(* POU Functions/F_GetVersionDehoff, ST *)
FUNCTION F_GetVersionDehoff : UINT
VAR_INPUT
	nVersionElement: INT := 0;
END_VAR
(*	Version history: This is for the program in the CX2020.  The HMI program version resisdes in the CP2612
Date	|	Rev	|	created under	|	Author				|	Remark		
---------------------------------------------------------------------------------------------------------------------------------------------------------------------
09/27/14	|	1.0	|	Build 2241	|	Ron Poehlmann		|	(Shipped on Machine #1 & 2)
12/04/14	|	1.1	|	Build 2241	|	Ron Poehlmann		|	Fixed problem caused by Fault History not being completed
															Added Fault Screen with Servo Axis Diagnostics #'s
															Moved into Persistent Data: U/X Axis Position and Speed variables & Tailstock Max Thrust
															Fixed Rung 117 to say 3B instead of 3A
															(* Remotely Installed on Machine #1 & #2*)
2/09/15	|	1.2	|	Build 2241	|	Ron Poehlmann		|	Changed Drill Cycle so that the Filter Fault does not stop the cycle.
															Worked on other Problems.
															(* Remotely Installed on Machine #2 & #1 *)
2/16/15	|	1.3	|	Build 2241	|	Ron Poehlmann		|	Rewrote Transfer Cycle.
															(* Remotely Installed on Machine #1 & #2 *)
2/18/15	|	1.3b	|											Fixed Reset of Servo Drives.
															(* Remotely Installed on Machine #1 & 2 *)
3/3/15	|	1.4	|	Build 2241	|	Ron Poehlmann		|	Added Recovery of Overtravel.
															Added checks and warnings before entering Auto.
															Added Single Homeing Button for WA, WB, and X Axis
															Modified Network Variables to assure alignment.
															Added Faults to Tailstock and Transfer.
															Shortened User name Passwords and added handshake bit.
															Added Recording of the W Axis Max Thrust Values.
															Added VFD Data Valid bit and Revised FB_EtherCAT_Emerson. 
7/8/15		Field mods										Added monitoring screen to CX to be able to view machie status.
															( Remotely Installed on Machine #1 - 4 )
11/05/15	|	1.5	|	Build 2241	|	Ron Poehlmann		|	Fixed typo that caused the X Axis Velocity not to be received from Panel B
															Added Fault condition to AC_CellRunoutFinish so it would Exit Auto on a Fault condition.
															Added Fault condition to AC_Init so it would Exit Auto on a Fault condition.
															Added Feed Over-ride as a setup feature.
															Fault at end of cycle if Lube Level Low Warning on for more than 2 cycles.
															Disable MPG if clamped.
															Fixed typo in FB_FixtureControl line 444 from nClampState to nUnclampState
															Changed Max Thrust Inputs for FB_Fixture Control
1/14/16	|	1.6	|	Build 2254	|	Ron Poehlmann		|	System Manager was Changed from V1 to V1.1 because of newer Card definitions.
															When Load Side switched - Swapp Load and unload Positions.
															Fixed a problem with the Waring 110 on Transfer_Cycle so that it will retriger in Cell Runout
																made step 10 check for bCellRunoutRequest.
*)
CASE nVersionElement OF
	1: F_GetVersionDehoff:=1;		(* Major Number *)
	2: F_GetVersionDehoff:=6;		(* ArboMex Program Revision Number *)
ELSE
	F_GetVersionDehoff:=16#FFFF;
END_CASE
END_FUNCTION

(* POU Programs/Build_Receive_Network_Data, ST *)
PROGRAM Build_Receive_Network_Data
VAR
	fbSideAUserNameInput: R_TRIG;			(* An User Name Input has just been received from Panel A *)
	fbSideBUserNameInput: R_TRIG;			(* An User Name Input has just been received from Panel B *)
	fbSideAPasswordInput: R_TRIG;				(* A Password Input has just been received from Panel A *)
	fbSideBPasswordInput: R_TRIG;				(* A Password Input has just been received from Panel B *)
	fbSideASavePasswordInputTrig: R_TRIG;		(* A Save Password Input has just been received from Panel A *)
	fbSideBSavePasswordInput: R_TRIG;		(* A Save Password Input has just been received from Panel B *)
	fbSideAEnableRTrig: R_TRIG;
	fbSideBEnableRTrig: R_TRIG;
	fbTestSpeedActiveRTrig: R_TRIG;			(* Push Button pressed to Activate/Deactivate the Test Speed *)
	nTest: INT := 0;		(* Test Counter*)
	fUAxisLoadPositionTempVariable: LREAL := 0.0;		(*A Temp variable used to swap the Load and unload position*)
END_VAR
(* Login Varialbes *)
(* If the Login PB or Logout PB is pressed on either screen, then turn on the bit*)
bLoginPB := stReceivePanelA.arrBOOL[8] OR stReceivePanelB.arrBOOL[8];
bLogoutPB := stReceivePanelA.arrBOOL[9] OR stReceivePanelB.arrBOOL[9];

(* Receive the User ID Input *)
(* Only place what is received into the Username when the received value first changes
	Also if they enter a wrong value, then we want to trigger when it changes. 
	When we see a change from '' set the handshake bit.  
		The Panel will then set the variable to '' again, so turn off the handshake bit.*)
fbSideAUserNameInput(CLK:=stReceivePanelA.arrTEXTSTRING[2] <> '');
fbSideBUserNameInput(CLK:=stReceivePanelB.arrTEXTSTRING[2] <> '');
IF fbSideAUserNameInput.Q THEN
	bUserNameHandshake:=TRUE;
	sUsername := stReceivePanelA.arrTEXTSTRING[2];
ELSIF fbSideBUserNameInput.Q THEN
	bUserNameHandshake:=TRUE;
	sUsername := stReceivePanelB.arrTEXTSTRING[2];
ELSIF (stReceivePanelA.arrTEXTSTRING[2] = '') AND (stReceivePanelB.arrTEXTSTRING[2] = '') THEN
	bUserNameHandshake:=FALSE;
END_IF

(* Receive the Password Input *)
fbSideAPasswordInput(CLK:=stReceivePanelA.arrTEXTSTRING[3] <> '');
fbSideBPasswordInput(CLK:=stReceivePanelB.arrTEXTSTRING[3] <> '');
IF fbSideAPasswordInput.Q THEN
	bPasswordHandshake:=TRUE;
	sPassword := stReceivePanelA.arrTEXTSTRING[3];
ELSIF fbSideBPasswordInput.Q THEN
	bPasswordHandshake:=TRUE;
	sPassword := stReceivePanelB.arrTEXTSTRING[3];
ELSIF (stReceivePanelA.arrTEXTSTRING[3] = '') AND (stReceivePanelB.arrTEXTSTRING[3] = '') THEN
	bPasswordHandshake:=FALSE;
END_IF

(* Receive the Save Password Input *)
fbSideASavePasswordInputTrig(CLK:=stReceivePanelA.arrTEXTSTRING[4] <> '');
fbSideBSavePasswordInput(CLK:=stReceivePanelB.arrTEXTSTRING[4] <> '');
IF (stReceivePanelA.arrTEXTSTRING[4] <> '') THEN
	IF stReceivePanelA.arrTEXTSTRING[4]=sPasswordSupervisorUC OR
		stReceivePanelA.arrTEXTSTRING[4]=sPasswordSupervisor OR
		stReceivePanelA.arrTEXTSTRING[4]=sPasswordSuperUC OR
		stReceivePanelA.arrTEXTSTRING[4]=sPasswordSuper
	THEN
		bWrongSavePassword:=FALSE;
		bSavePasswordHandshake:=TRUE;
		sSavePassword := stReceivePanelA.arrTEXTSTRING[4];
	(* Password is not correct *)
	ELSE
		bWrongSavePassword:=TRUE;
	END_IF
END_IF
IF (stReceivePanelB.arrTEXTSTRING[4] <> '') THEN
	IF stReceivePanelB.arrTEXTSTRING[4]=sPasswordSupervisorUC OR
		stReceivePanelB.arrTEXTSTRING[4]=sPasswordSupervisor OR
		stReceivePanelA.arrTEXTSTRING[4]=sPasswordSuperUC OR
		stReceivePanelA.arrTEXTSTRING[4]=sPasswordSuper
	THEN
		bWrongSavePassword:=FALSE;
		bSavePasswordHandshake:=TRUE;
		sSavePassword := stReceivePanelB.arrTEXTSTRING[4];
		(* Password is not correct *)
	ELSE
		bWrongSavePassword:=TRUE;
	END_IF
END_IF
IF (stReceivePanelA.arrTEXTSTRING[4] = '') AND (stReceivePanelB.arrTEXTSTRING[4] = '') THEN
	bSavePasswordHandshake:=FALSE;
	bWrongSavePassword:=FALSE;
END_IF


(* Call Actions *)
Auto_Screen_Receive;
Part_Program_Screen;
Transfer_Screen;
Fixture_Screen;
Secret_Screen;
Test_Speed_Screen;
Manual_Screen_Receive;
END_PROGRAM
ACTION Auto_Screen_Receive:
(* Push Buttons *)
bEnterManualModePB := 	stReceivePanelA.arrBOOL[1] OR stReceivePanelB.arrBOOL[1];
bEnterAutoModePB := 		stReceivePanelA.arrBOOL[2] OR stReceivePanelB.arrBOOL[2];
bResetCycleCounterPB := 	stReceivePanelA.arrBOOL[3] OR stReceivePanelB.arrBOOL[3];;
bFaultResetPB := 			stReceivePanelA.arrBOOL[4] OR stReceivePanelB.arrBOOL[4];
bResetTotalCountPB := 	stReceivePanelA.arrBOOL[5] OR stReceivePanelB.arrBOOL[5];
bCellRunOutPB := 			stReceivePanelA.arrBOOL[67] OR stReceivePanelB.arrBOOL[67];
bResetA1CountPB:= 		stReceivePanelA.arrBOOL[42] OR stReceivePanelB.arrBOOL[42];
bResetA2CountPB:= 		stReceivePanelA.arrBOOL[43] OR stReceivePanelB.arrBOOL[43];
bResetA3CountPB:= 		stReceivePanelA.arrBOOL[44] OR stReceivePanelB.arrBOOL[44];
bResetB1CountPB:= 		stReceivePanelA.arrBOOL[45] OR stReceivePanelB.arrBOOL[45];
bResetB2CountPB:= 		stReceivePanelA.arrBOOL[46] OR stReceivePanelB.arrBOOL[46];
bResetB3CountPB:= 		stReceivePanelA.arrBOOL[47] OR stReceivePanelB.arrBOOL[47];
END_ACTION
ACTION Fixture_Screen:
(* Fixture common Inputs *)
(* When a Transfer position Input is received from Panel A or B then modify *)
IF stReceivePanelA.arrLREAL[20] <> 0.0 THEN
	fWAxisTransferPosition :=stReceivePanelA.arrLREAL[20];
ELSIF stReceivePanelB.arrLREAL[20] <> 0.0 THEN
	fWAxisTransferPosition :=stReceivePanelB.arrLREAL[20];
END_IF

(* When a Drill Position Input is received from Panel A or B then modify *)
IF stReceivePanelA.arrLREAL[21] <> 0.0 THEN
	fWAxisDrillPosition :=stReceivePanelA.arrLREAL[21];
ELSIF stReceivePanelB.arrLREAL[21] <> 0.0 THEN
	fWAxisDrillPosition :=stReceivePanelB.arrLREAL[21];
END_IF

(* A Side *)
(*Push Buttons Side A *)
bWAAxisHomePB := stReceivePanelA.arrBOOL[30];
bWAAxisAdvancePB := stReceivePanelA.arrBOOL[31];
bWAAxisRetractPB := stReceivePanelA.arrBOOL[32];
bAColletClosePB := stReceivePanelA.arrBOOL[33];
bAColletOpenPB := stReceivePanelA.arrBOOL[34];
bAEjectorsAdvancePB := stReceivePanelA.arrBOOL[35];
bAEjectorsRetractPB := stReceivePanelA.arrBOOL[36];

	(* B Side *)
(*Push Buttons Side B *)
bWBAxisHomePB := stReceivePanelB.arrBOOL[30];
bWBAxisAdvancePB := stReceivePanelB.arrBOOL[31];
bWBAxisRetractPB := stReceivePanelB.arrBOOL[32];
bBColletClosePB := stReceivePanelB.arrBOOL[33];
bBColletOpenPB := stReceivePanelB.arrBOOL[34];
bBEjectorsAdvancePB := stReceivePanelB.arrBOOL[35];
bBEjectorsRetractPB := stReceivePanelB.arrBOOL[36];

(* If We have a FAULT we do not want to permit manual operations.
	So turn off any PB bits that may have been pushed. *)
IF bMachineFault
	OR nAutoCycleStep=AC_Drill
	OR nAutoCycleStep=AC_DrillReturn
	OR nAutoCycleStep=AC_Retract
THEN
	bWAAxisHomePB := FALSE;
	bWAAxisAdvancePB := FALSE;
	bWAAxisRetractPB := FALSE;
	bAColletClosePB := FALSE;
	bAColletOpenPB := FALSE;
	bAEjectorsAdvancePB := FALSE;
	bAEjectorsRetractPB := FALSE;
	bWBAxisHomePB := FALSE;
	bWBAxisAdvancePB := FALSE;
	bWBAxisRetractPB := FALSE;
	bBColletClosePB := FALSE;
	bBColletOpenPB := FALSE;
	bBEjectorsAdvancePB := FALSE;
	bBEjectorsRetractPB := FALSE;
END_IF
END_ACTION
ACTION Manual_Screen_Receive:
(* MANUAL SCREEN *)

(* Push Buttons *)
(* When the Start Hydraulic PB is pressed on either panel *)
bStartHydraulicPB := stReceivePanelA.arrBOOL[60] OR stReceivePanelB.arrBOOL[60];
(* When the Stop Hydraulic PB is pressed on either panel *)
bStopHydraulicPB := stReceivePanelA.arrBOOL[61] OR stReceivePanelB.arrBOOL[61];
(* When the Start Coolant PB is pressed on either panel *)
bCoolantStartPB := stReceivePanelA.arrBOOL[62] OR stReceivePanelB.arrBOOL[62];
(* When the Stop Coolant PB is pressed on either panel *)
bCoolantStopPB := stReceivePanelA.arrBOOL[63] OR stReceivePanelB.arrBOOL[63];
(* Setup is dependant on the side it is Pressed *)
bEnterSetupPB_A := stReceivePanelA.arrBOOL[64];
bEnterSetupPB_B := stReceivePanelB.arrBOOL[64];
(* Set Zero is dependant on the side it is Pressed *)
bSetZeroPositionPB_A := stReceivePanelA.arrBOOL[65];
bSetZeroPositionPB_B := stReceivePanelB.arrBOOL[65];
(* Move To Zero is dependant on the side it is Pressed *)
bMoveToZeroPositionPB_A := stReceivePanelA.arrBOOL[66];
bMoveToZeroPositionPB_B := stReceivePanelB.arrBOOL[66];

(* When the Home All Automation PB is pressed on either panel *)
bHomeAutomationPB := stReceivePanelA.arrBOOL[68] OR stReceivePanelB.arrBOOL[68];
END_ACTION
ACTION Part_Program_Screen:
(* PART PROGRAM Inputs *)

(*  Change the Part Program Name when Inserted by operator *)
IF stReceivePanelA.arrTEXTSTRING[1] <> ''  THEN
	sPartProgramName := stReceivePanelA.arrTEXTSTRING[1];
ELSIF stReceivePanelB.arrTEXTSTRING[1] <> '' THEN
	sPartProgramName := stReceivePanelB.arrTEXTSTRING[1];
END_IF

(* Save Part Progarm Push Button *)
bPartProgramSavePB:= stReceivePanelA.arrBOOL[11] OR stReceivePanelB.arrBOOL[11];

(* Leave the PP_SAVE screen *)
IF stReceivePanelA.arrBOOL[69] OR stReceivePanelB.arrBOOL[69] THEN
	sSavePassword:='';
END_IF


(* Load Part Program Push Button - Not available in Auto  *)
bPartProgramLoadPB := stReceivePanelA.arrBOOL[12] OR stReceivePanelB.arrBOOL[12];

(**** IMPORTANT! ***  If the system is in AUTO or In Cycle we need to send a Warning  *)

(* Toggle the state of Spindle Retract mode when PB received from panels *)
IF stReceivePanelA.arrBOOL[10] OR stReceivePanelB.arrBOOL[10] THEN
	IF bSpindleRetractMode THEN
		bSpindleRetractMode:=FALSE;
	ELSE bSpindleRetractMode:=TRUE;
	END_IF
END_IF

(* When a Start Feed Input is received from either panel then modify *)
IF stReceivePanelA.arrLREAL[1] > 0.0 THEN
	fStartFeed:=stReceivePanelA.arrLREAL[1];
ELSIF stReceivePanelB.arrLREAL[1] > 0.0 THEN
	fStartFeed:=stReceivePanelB.arrLREAL[1];
END_IF

(* When a Start Feed Input is received from either panel then modify *)
IF stReceivePanelA.arrLREAL[2] > 0.0 THEN
	fFinishFeed:=stReceivePanelA.arrLREAL[2];
ELSIF stReceivePanelB.arrLREAL[2] > 0.0 THEN
	fFinishFeed:=stReceivePanelB.arrLREAL[2];
END_IF

(* When a Start Depth Input is received from either panel then modify *)
IF stReceivePanelA.arrLREAL[3] < 0.0 THEN
	fStartDepth:=stReceivePanelA.arrLREAL[3];
ELSIF stReceivePanelB.arrLREAL[3] < 0.0 THEN
	fStartDepth:=stReceivePanelB.arrLREAL[3];
END_IF

(* When a Finish Depth Input is received from either panel then modify *)
IF stReceivePanelA.arrLREAL[4] < 0.0 THEN
	fFinishDepth:=stReceivePanelA.arrLREAL[4];
ELSIF stReceivePanelB.arrLREAL[4] < 0.0 THEN
	fFinishDepth:=stReceivePanelB.arrLREAL[4];
END_IF

(* When a Dwell Time Input is received from either panel then modify *)
IF stReceivePanelA.arrLREAL[5] > 0.0 THEN
	fDwellTime:=stReceivePanelA.arrLREAL[5];
ELSIF stReceivePanelB.arrLREAL[5] > 0.0 THEN
	fDwellTime:=stReceivePanelB.arrLREAL[5];
END_IF

(* When a Retract Rate Input is received from either panel then modify *)
IF stReceivePanelA.arrLREAL[6] > 0.0 THEN
	fRetractRate:=stReceivePanelA.arrLREAL[6];
ELSIF stReceivePanelB.arrLREAL[6] > 0.0 THEN
	fRetractRate:=stReceivePanelB.arrLREAL[6];
END_IF

(* When a fDrill Tip Offset Input is received from either panel then modify *)
IF stReceivePanelA.arrLREAL[7] > 0.0 THEN
	fDrillTipOffset:=stReceivePanelA.arrLREAL[7];
ELSIF stReceivePanelB.arrLREAL[7] > 0.0 THEN
	fDrillTipOffset:=stReceivePanelB.arrLREAL[7];
END_IF

(* When a RPM Request Input is received from either panel then modify *)
IF stReceivePanelA.arrLREAL[8] > 0.0 THEN
	fRPMRequest:=stReceivePanelA.arrLREAL[8];
ELSIF stReceivePanelB.arrLREAL[8] > 0.0 THEN
	fRPMRequest:=stReceivePanelB.arrLREAL[8];
END_IF

(* When a Tool Diameter Input is received from either panel then modify *)
IF stReceivePanelA.arrLREAL[9] > 0.0 THEN
	fToolDiameter:=stReceivePanelA.arrLREAL[9];
ELSIF stReceivePanelB.arrLREAL[9] > 0.0 THEN
	fToolDiameter:=stReceivePanelB.arrLREAL[9];
END_IF

(* When a Coolant Pressure Input is received from either panel then modify *)
IF stReceivePanelA.arrLREAL[10] > 0.0 THEN
	fCoolantPressure:=stReceivePanelA.arrLREAL[10];
ELSIF stReceivePanelB.arrLREAL[10] > 0.0 THEN
	fCoolantPressure:=stReceivePanelB.arrLREAL[10];
END_IF

(* When a Coolant Flow Max Input is received from either panel then modify *)
IF stReceivePanelA.arrLREAL[11] > 0.0 THEN
	fCoolantFlowMax:=stReceivePanelA.arrLREAL[11];
ELSIF stReceivePanelB.arrLREAL[11] > 0.0 THEN
	fCoolantFlowMax:=stReceivePanelB.arrLREAL[11];
END_IF

(* When a Coolant Flow Min Input is received from either panel then modify *)
IF stReceivePanelA.arrLREAL[12] > 0.0 THEN
	fCoolantFlowMin:=stReceivePanelA.arrLREAL[12];
ELSIF stReceivePanelB.arrLREAL[12] > 0.0 THEN
	fCoolantFlowMin:=stReceivePanelB.arrLREAL[12];
END_IF

(* When Max cycles Set is received from either panel then modify *)
IF stReceivePanelA.arrUDINTIGER[1] > 0 THEN
	nMaxCycles := stReceivePanelA.arrUDINTIGER[1];
ELSIF  stReceivePanelB.arrUDINTIGER[1] > 0 THEN
	nMaxCycles := stReceivePanelB.arrUDINTIGER[1];
END_IF

(* When Spindle Load Max Set is received from either panel then modify *)
IF stReceivePanelA.arrUDINTIGER[2] > 0 THEN
	nSpindleLoadMax := stReceivePanelA.arrUDINTIGER[2];
ELSIF  stReceivePanelB.arrUDINTIGER[2] > 0 THEN
	nSpindleLoadMax := stReceivePanelB.arrUDINTIGER[2];
END_IF

(* When Servo Thrust Max Set is received from either panel then modify *)
IF stReceivePanelA.arrUDINTIGER[3] > 0 THEN
	nServoThrustMax := stReceivePanelA.arrUDINTIGER[3];
ELSIF  stReceivePanelB.arrUDINTIGER[3] > 0 THEN
	nServoThrustMax := stReceivePanelB.arrUDINTIGER[3];
END_IF
END_ACTION
ACTION Secret_Screen:
(* Receive the PB's from the Panels *)
(* The Panels Make sure you must not be in Auto Mode *)
IF stReceivePanelA.arrBOOL[6] OR stReceivePanelB.arrBOOL[6] THEN
	bASideIsLoadPB := TRUE;
ELSIF  stReceivePanelA.arrBOOL[7] OR stReceivePanelB.arrBOOL[7] THEN
	bBSideIsLoadPB := TRUE;
END_IF

fbSideAEnableRTrig(CLK:=stReceivePanelA.arrBOOL[40] OR stReceivePanelB.arrBOOL[40]);
IF fbSideAEnableRTrig.Q THEN
	IF bSideAEnabled THEN
		bSideAEnabled := FALSE;
	ELSE
		bSideAEnabled :=TRUE;
	END_IF
END_IF

fbSideBEnableRTrig(CLK:=stReceivePanelA.arrBOOL[41] OR stReceivePanelB.arrBOOL[41]);
IF fbSideBEnableRTrig.Q THEN
	IF bSideBEnabled THEN
		bSideBEnabled := FALSE;
	ELSE
		bSideBEnabled :=TRUE;
	END_IF
END_IF

IF bASideIsLoadPB THEN
	sLoadSideSet := 'A';
	(* Swap the Load and Unload Positions *)
	fUAxisLoadPositionTempVariable:=fUAxisLoadSidePosition;
	fUAxisLoadSidePosition:= fUAxisUnloadSidePosition;
	fUAxisUnloadSidePosition:=fUAxisLoadPositionTempVariable;
	bASideIsLoadPB := FALSE;
ELSIF bBSideIsLoadPB THEN
	sLoadSideSet :='B';
	(* Swap the Load and Unload Positions *)
	fUAxisLoadPositionTempVariable:=fUAxisLoadSidePosition;
	fUAxisLoadSidePosition:= fUAxisUnloadSidePosition;
	fUAxisUnloadSidePosition:=fUAxisLoadPositionTempVariable;
	bBSideIsLoadPB := FALSE;
END_IF

IF (stReceivePanelA.arrUDINTIGER[10] >0) THEN
	nUAxisThrustMax := stReceivePanelA.arrUDINTIGER[10];
ELSIF (stReceivePanelB.arrUDINTIGER[10] >0) THEN
	nUAxisThrustMax := stReceivePanelB.arrUDINTIGER[10];
END_IF

(* Tailstock Torque Limit During Clamping *)
IF (stReceivePanelA.arrUDINTIGER[11] >0) THEN
	nTailstockClampingTorqueLimit := UDINT_TO_INT(stReceivePanelA.arrUDINTIGER[11]);
ELSIF (stReceivePanelB.arrUDINTIGER[11] >0) THEN
	nTailstockClampingTorqueLimit := UDINT_TO_INT(stReceivePanelB.arrUDINTIGER[11]);
END_IF

(* Receive the WA Axis Home Offset *)
(* Must compare with current value because 0.0 is an option *)
IF stReceivePanelA.arrLREAL[17] <> 0.0  THEN
	fWAAxisHomeOffset := stReceivePanelA.arrLREAL[17];
ELSIF stReceivePanelB.arrLREAL[17] <> 0.0 THEN
	fWAAxisHomeOffset := stReceivePanelB.arrLREAL[17];
END_IF

(* Receive the WB Axis Home Offset *)
IF stReceivePanelA.arrLREAL[18] <> 0.0  THEN
	fWBAxisHomeOffset := stReceivePanelA.arrLREAL[18];
ELSIF stReceivePanelB.arrLREAL[18] <> 0.0 THEN
	fWBAxisHomeOffset := stReceivePanelB.arrLREAL[18];
END_IF

(* Receive the W Axis Amount to Move Off of Bushing *)
IF stReceivePanelA.arrLREAL[19] <> 0.0 THEN
	fWAxisMoveOffBushing :=stReceivePanelA.arrLREAL[19];
ELSIF stReceivePanelB.arrLREAL[19] <> 0.0 THEN
	fWAxisMoveOffBushing :=stReceivePanelB.arrLREAL[19];
END_IF

(* Receive the W Axis Move Velocity *)
IF stReceivePanelA.arrLREAL[24] > 0.0 THEN
	fTailstockVelocity :=stReceivePanelA.arrLREAL[24];
ELSIF stReceivePanelB.arrLREAL[24] > 0.0 THEN
	fTailstockVelocity :=stReceivePanelB.arrLREAL[24];
END_IF

(* When a WA Axis Max Thrust Input is received from Panel A then modify *)
IF stReceivePanelA.arrUDINTIGER[5] > 0.0 THEN
	nWAAxisThrustMax :=stReceivePanelA.arrUDINTIGER[5];
ELSIF stReceivePanelB.arrUDINTIGER[5] > 0.0 THEN
	nWAAxisThrustMax :=stReceivePanelB.arrUDINTIGER[5];
END_IF

(* When a WB Axis Max Thrust Input is received from Panel B then modify *)
IF stReceivePanelA.arrUDINTIGER[6] > 0.0 THEN
	nWBAxisThrustMax :=stReceivePanelA.arrUDINTIGER[6];
ELSIF stReceivePanelB.arrUDINTIGER[6] > 0.0 THEN
	nWBAxisThrustMax :=stReceivePanelB.arrUDINTIGER[6];
END_IF
END_ACTION
ACTION Test_Speed_Screen:
(* Test Speed  Screen *)
(* The Test Speed would be like a feed over-ride and changes the speeds of the WA, WB and X Axis movements *)

(* When either panel sets the  "Test Speed Input" then make it Current Test Speed *)
IF (stReceivePanelA.arrUDINTIGER[15] <> 0.0) THEN
	nTestSpeedOverRide := stReceivePanelA.arrUDINTIGER[15];
ELSIF (stReceivePanelB.arrUDINTIGER[15] <> 0.0) THEN
	nTestSpeedOverRide := stReceivePanelB.arrUDINTIGER[15];
END_IF

(* When the Test Speed Overide PB is pressed on either screen, we toggle the state On/Off *)
fbTestSpeedActiveRTrig(CLK:=stReceivePanelA.arrBOOL[15] OR stReceivePanelB.arrBOOL[15]);
IF fbTestSpeedActiveRTrig.Q THEN
	IF bTestSpeedOn THEN
		bTestSpeedOn := FALSE;
	ELSE
		bTestSpeedOn := TRUE;
	END_IF
END_IF

(* When the Test Speed is Activated we want to Change the velocities that we feed to the Axis Move FB's *)
IF bTestSpeedOn THEN
	fWAxisFastVelocity := fTailstockVelocity * (nTestSpeedOverRide/100.0);
	fWAxisClampVelocity :=  fTailstockClampVelocity * (nTestSpeedOverRide/100.0);
	fTransferMoveVelo := fUAxisVelocity  * (nTestSpeedOverRide/100.0);
ELSE
	fWAxisFastVelocity := fTailstockVelocity;
	fWAxisClampVelocity :=  fTailstockClampVelocity;
	fTransferMoveVelo:=  fUAxisVelocity;
END_IF
END_ACTION
ACTION Transfer_Screen:
(* TRANSFER Screen Inputs *)

(* Raise and Lower Push Buttons *)
bTransferUpPB := (stReceivePanelA.arrBOOL[20] OR stReceivePanelB.arrBOOL[20]);
bTransferDownPB := (stReceivePanelA.arrBOOL[21] OR stReceivePanelB.arrBOOL[21]);

(* Home U Axis PB *)
bHomeUAxisPB := (stReceivePanelA.arrBOOL[22] OR stReceivePanelB.arrBOOL[22]);

(* Move U Axis PB's *)
bMoveUtoLoadPB := (stReceivePanelA.arrBOOL[23] OR stReceivePanelB.arrBOOL[23]);
bMoveUtoUnloadPB := (stReceivePanelA.arrBOOL[24] OR stReceivePanelB.arrBOOL[24]);

(* When we have a FAULT we want to disable manual functions.
	So turn off any PB's that could have been pushed *) 
IF bMachineFault
	OR nAutoCycleStep=AC_Drill
	OR nAutoCycleStep=AC_DrillReturn
	OR nAutoCycleStep=AC_Retract
THEN
	bTransferUpPB := FALSE;
	bTransferDownPB := FALSE;
	bHomeUAxisPB:= FALSE;
	bMoveUtoLoadPB:= FALSE;
	bMoveUtoUnloadPB:= FALSE;
END_IF

(* When either side sets the U Axis A Side position then put it in appropriate Load or Unload variable *)
IF (stReceivePanelA.arrLREAL[15] <>0) THEN	(* fUAxisASidePositionInput *)
	IF (sLoadSideSet = 'A') THEN
		fUAxisLoadSidePosition := stReceivePanelA.arrLREAL[15];
	ELSIF (sLoadSideSet = 'B') THEN
		fUAxisUnloadSidePosition := stReceivePanelA.arrLREAL[15];
	ELSE
		bLoadSideNotSelected := TRUE;
	END_IF
ELSIF (stReceivePanelB.arrLREAL[15] <>0) THEN	(* fUAxisASidePositionInput *)
	IF (sLoadSideSet = 'A') THEN
		fUAxisLoadSidePosition := stReceivePanelB.arrLREAL[15];
	ELSIF (sLoadSideSet = 'B') THEN
		fUAxisUnloadSidePosition := stReceivePanelB.arrLREAL[15];
	ELSE
		bLoadSideNotSelected := TRUE;
	END_IF
END_IF

(* When either side sets the U Axis B Side position then put it in appropriate Load or Unload variable *)
IF (stReceivePanelA.arrLREAL[16] <> 0.0) THEN	(* fUAxisBSidePositionInput *)
	IF (sLoadSideSet = 'A') THEN
		fUAxisUnloadSidePosition := stReceivePanelA.arrLREAL[16];
	ELSIF (sLoadSideSet = 'B') THEN
		fUAxisLoadSidePosition := stReceivePanelA.arrLREAL[16];
	ELSE
		bLoadSideNotSelected := TRUE;
	END_IF
ELSIF (stReceivePanelB.arrLREAL[16] <> 0.0) THEN	(* fUAxisBSidePositionInput *)
	IF (sLoadSideSet = 'A') THEN
		fUAxisUnloadSidePosition := stReceivePanelB.arrLREAL[16];
	ELSIF (sLoadSideSet = 'B') THEN
		fUAxisLoadSidePosition := stReceivePanelB.arrLREAL[16];
	ELSE
		bLoadSideNotSelected := TRUE;
	END_IF
END_IF

(* When either side sets the U Axis "Transfer Speed" then make it Current Speed *)
IF (stReceivePanelA.arrLREAL[25] <> 0.0) THEN
	fUAxisVelocity := stReceivePanelA.arrLREAL[25];
ELSIF (stReceivePanelB.arrLREAL[25] <> 0.0) THEN
	fUAxisVelocity := stReceivePanelB.arrLREAL[25];
END_IF
END_ACTION

(* POU Programs/P_PartProgramStorage, ST *)
PROGRAM P_PartProgramStorage
VAR
	fbPartProgramSaveRTRIG: R_TRIG;			(* Trigger for Part Program Save PB *)
	fbPartProgramLoadRTRIG: R_TRIG;			(* Trigger for Part Program Load PB *)
	bSave: BOOL := FALSE;
	bLoad: BOOL := FALSE;
	bFailed: BOOL := FALSE;
	bSuccess: BOOL := FALSE;

	(* Function Blocks w/ Helpers *)
	fbFileOpen: FB_FileOpen;
	bFileOpen: BOOL := FALSE;
	fbFileClose: FB_FileClose;
	nOpenType: DWORD;
	bFileClose: BOOL := FALSE;
	fbFilePuts: FB_FilePuts;
	bFilePuts: BOOL := FALSE;
	fbFileGets: FB_FileGets;
	bFileGets: BOOL := FALSE;
	hFileHandle: UINT := 0;
	sFileName: T_MaxString := '';

	(* State Variables *)
	nStep: USINT := 0;

	(* Read Variables  Note: if size changes it must be changed here and in the program below *)
	arrDataRead: ARRAY [1..25] OF T_MaxString;
	nReadCount: USINT := 0;

	(* Write Variables *)
	arrDataWrite: ARRAY [1..25] OF T_MaxString;
	nWriteCount: USINT := 0;

	nTestCount: INT := 0;		(* Test Counter *)
	bTestbit1: BOOL := FALSE;		(* Test Bit *)
END_VAR
fbPartProgramSaveRTRIG(CLK:= bPartProgramSavePB);
fbPartProgramLoadRTRIG(CLK:= bPartProgramLoadPB);

IF fbPartProgramSaveRTRIG.Q AND NOT(bSave OR bLoad) THEN
	(* When the Yes PB is pressed then check the password input *)
	IF sSavePassword=sPasswordSupervisorUC OR
		sSavePassword=sPasswordSupervisor OR
		sSavePassword=sPasswordSuperUC OR
		sSavePassword=sPasswordSuper
	THEN	(* Reset Values *)
		bFailed:=FALSE;
		bSuccess:=FALSE;
		sFileOpError:='';
		bSave:=TRUE;
		sSavePassword:='';
	END_IF
ELSIF fbPartProgramLoadRTRIG.Q AND NOT(bSave OR bLoad) THEN
	bFailed:=FALSE;
	sFileOpError:='';
	bSuccess:=FALSE;
	bLoad:=TRUE;
END_IF

sFileName:=CONCAT('\Hard Disk\ftp\',CONCAT(sPartProgramName, '.CSV'));


(* Load Part Program *)
IF bLoad AND NOT(bSave) THEN
	CASE nStep OF
	0:(* Open File *)
		nOpenType:=FOPEN_MODEREAD;
		(*ERROR*)
		IF bFileOpen AND fbFileOpen.bError THEN
			bFileOpen:=FALSE;
			bLoad:=FALSE;
			bFailed:=TRUE;
			sFileOpError:=CONCAT('Open Error:  ',UDINT_TO_STRING(fbFileOpen.nErrId));
		ELSIF bFileOpen AND NOT(fbFileOpen.bBusy) THEN
			bFileOpen:=FALSE;
			nReadCount:=1;
			nStep:=nStep+1;
		END_IF
		bFileOpen:=TRUE;

	1:(* Read File *)
		IF (nReadCount<=25) OR NOT(fbFileGets.bEOF) THEN
			(*ERROR*)
			IF bFileGets AND fbFileGets.bError THEN
				nStep:=nStep+1;
				bFailed:=TRUE;
				sFileOpError:=CONCAT('Read Error:  ',UDINT_TO_STRING(fbFileGets.nErrId));
			ELSIF bFileGets AND NOT(fbFileGets.bBusy) THEN
				arrDataRead[nReadCount]:=fbFileGets.sLine;
				bFileGets:=FALSE;
				nReadCount:=nReadCount+1;
			ELSIF NOT(bFileGets) THEN
				bFileGets:=TRUE;
			END_IF
		END_IF
		IF nReadCount>25 THEN
			nStep:=nStep+1;
		END_IF

	2:(* Close File *)
		(*ERROR*)
		IF bFileClose AND fbFileClose.bError THEN
			sFileOpError:=CONCAT('Close Error:  ',UDINT_TO_STRING(fbFileClose.nErrId));
			bFileClose:=FALSE;
			bLoad:=FALSE;
			bFailed:=TRUE;
		ELSIF bFileClose AND NOT(fbFileClose.bBusy) THEN
			bFileClose:=FALSE;
			IF bFailed THEN
				bLoad:=FALSE;
			ELSE
				nStep:=nStep+1;
			END_IF
		END_IF
		bFileClose:=TRUE;

	3:(* Convert Data / Done *)
		fStartFeed				:= STRING_TO_LREAL(arrDataRead[2]);
		fFinishFeed 				:= STRING_TO_LREAL(arrDataRead[3]);
		fStartDepth 				:= STRING_TO_LREAL(arrDataRead[4]);
		fFinishDepth 				:= STRING_TO_LREAL(arrDataRead[5]);
		fDwellTime 				:= STRING_TO_LREAL(arrDataRead[6]);
		fRetractRate 				:= STRING_TO_LREAL(arrDataRead[7]);
		fDrillTipOffset				:= STRING_TO_LREAL(arrDataRead[8]);
		fRPMRequest			:= STRING_TO_LREAL(arrDataRead[9]);
		fToolDiameter			:= STRING_TO_LREAL(arrDataRead[10]);
		fCoolantPressure			:= STRING_TO_LREAL(arrDataRead[11]);
		fCoolantFlowMax			:= STRING_TO_LREAL(arrDataRead[12]);
		fCoolantFlowMin			:= STRING_TO_LREAL(arrDataRead[13]);
		nMaxCycles				:= LREAL_TO_UDINT(STRING_TO_LREAL(arrDataRead[14]));
		fWAxisTransferPosition		:= STRING_TO_LREAL(arrDataRead[15]);
		fWAxisDrillPosition		:= STRING_TO_LREAL(arrDataRead[16]);
		fWAxisMoveOffBushing		:= STRING_TO_LREAL(arrDataRead[17]);
		(*	:= STRING_TO_LREAL(arrDataRead[18]);		*)
		bSpindleRetractMode		:= STRING_TO_BOOL(arrDataRead[19]);
		nSpindleLoadMax			:= LREAL_TO_UDINT(STRING_TO_LREAL(arrDataRead[20]));
		nServoThrustMax			:= LREAL_TO_UDINT(STRING_TO_LREAL(arrDataRead[21]));
		(*	:=STRING_TO_LREAL(arrDataRead[22]);		*)
		(*	:=STRING_TO_LREAL(arrDataRead[23]);		*)
		(*	:=STRING_TO_LREAL(arrDataRead[24]);		*)
		(*	:=STRING_TO_LREAL(arrDataRead[25]);		*)
		(* IF MORE THAN 25 VARIABLES
			THEN MUST CHANGE nReadCount COMPARASONS IN nStep 1 *)
		nStep:=nStep+1;

	4:(* Done *)
		nStep:=0;
		bLoad:=FALSE;
		bSuccess:=TRUE;
		sLastLoadedPartProgramName := sPartProgramName;
		sCurrentPartProgram := sPartProgramName;

	END_CASE


ELSIF bSave AND NOT(bLoad) THEN
	CASE nStep OF
	0:(* Prepare Data *)
		arrDataWrite[1]	:= CONCAT(sPartProgramName,'$L');
		arrDataWrite[2]	:= CONCAT(LREAL_TO_STRING(fStartFeed),'$L');
		arrDataWrite[3]	:= CONCAT(LREAL_TO_STRING(fFinishFeed),'$L');
		arrDataWrite[4]	:= CONCAT(LREAL_TO_STRING(fStartDepth),'$L');
		arrDataWrite[5]	:= CONCAT(LREAL_TO_STRING(fFinishDepth),'$L');
		arrDataWrite[6]	:= CONCAT(LREAL_TO_STRING(fDwellTime),'$L');
		arrDataWrite[7]	:= CONCAT(LREAL_TO_STRING(fRetractRate),'$L');
		arrDataWrite[8]	:= CONCAT(LREAL_TO_STRING(fDrillTipOffset),'$L');
		arrDataWrite[9]	:= CONCAT(LREAL_TO_STRING(fRPMRequest),'$L');
		arrDataWrite[10]	:= CONCAT(LREAL_TO_STRING(fToolDiameter),'$L');
		arrDataWrite[11]	:= CONCAT(LREAL_TO_STRING(fCoolantPressure),'$L');
		arrDataWrite[12]	:= CONCAT(LREAL_TO_STRING(fCoolantFlowMax),'$L');
		arrDataWrite[13]	:= CONCAT(LREAL_TO_STRING(fCoolantFlowMin),'$L');
		arrDataWrite[14]	:= CONCAT(UDINT_TO_STRING(nMaxCycles),'$L');
		arrDataWrite[15]	:= CONCAT(LREAL_TO_STRING(fWAxisTransferPosition),'$L');
		arrDataWrite[16]	:= CONCAT(LREAL_TO_STRING(fWAxisDrillPosition),'$L');
		arrDataWrite[17]	:= CONCAT(LREAL_TO_STRING(fWAxisMoveOffBushing),'$L');
		arrDataWrite[18]	:= '$L';
		arrDataWrite[19]	:= CONCAT(BOOL_TO_STRING(bSpindleRetractMode),'$L');
		arrDataWrite[20]	:= CONCAT(UDINT_TO_STRING(nSpindleLoadMax),'$L');
		arrDataWrite[21]	:= CONCAT(UDINT_TO_STRING(nServoThrustMax),'$L');
		arrDataWrite[22]	:= '$L';
		arrDataWrite[23]	:= '$L';
		arrDataWrite[24]	:= '$L';
		arrDataWrite[25]	:= '$L';
		(* IF MORE THAN 25 VARIABLES
			THEN MUST CHANGE nReadCount COMPARASONS IN nStep 1 *)
		nStep:=nStep+1;

	1:(* Open File *)
		nOpenType:=FOPEN_MODEWRITE;
		(*ERROR*)
		IF bFileOpen AND fbFileOpen.bError THEN
			bFileOpen:=FALSE;
			bSave:=FALSE;
			bFailed:=TRUE;
			sFileOpError:=CONCAT('Open Error:  ',UDINT_TO_STRING(fbFileOpen.nErrId));
		ELSIF bFileOpen AND NOT(fbFileOpen.bBusy) THEN
			bFileOpen:=FALSE;
			nWriteCount:=1;
			nStep:=nStep+1;
		END_IF
		bFileOpen:=TRUE;

	2:(* Write File *)
		(* Wrie the string from the array until we write all of the data *)
		IF (nWriteCount<=25) THEN
			(*ERROR*)
			IF bFilePuts AND fbFilePuts.bError THEN
				nStep:=nStep+1;
				bFailed:=TRUE;
				sFileOpError:=CONCAT('WriteError:  ',UDINT_TO_STRING(fbFilePuts.nErrId));
			(* when no longer bussy then we incriment the count *)
			ELSIF bFilePuts AND NOT(fbFilePuts.bBusy) THEN
				bFilePuts:=FALSE;
				nWriteCount:=nWriteCount+1;
			(* Push the next value into the line and trigger the move (fileputs) *)
			ELSIF NOT(bFilePuts) THEN
				fbFilePuts.sLine:=arrDataWrite[nWriteCount];
				bFilePuts:=TRUE;
			END_IF
		(* Once we've put all of the date into the file we move to the next step *)
		ELSIF nWriteCount>25 THEN
			nStep:=nStep+1;
		END_IF
;
	3:(* Close File *)
		(*ERROR*)
		IF bFileClose AND fbFileClose.bError THEN
			bFileClose:=FALSE;
			bSave:=FALSE;
			bFailed:=TRUE;
			sFileOpError:=CONCAT('Close Error:  ',UDINT_TO_STRING(fbFileClose.nErrId));
		ELSIF bFileClose AND NOT(fbFileClose.bBusy) THEN
			IF NOT(bFailed) THEN
				bSuccess:=TRUE;
			END_IF
			bFileClose:=FALSE;
			bSave:=FALSE;
			nStep:=0;
		END_IF
		bFileClose:=TRUE;

	END_CASE

ELSE (* Not bLoad or bSave *)
	nStep:=0;
	nReadCount:=0;
	nWriteCount:=0;
	bFileOpen:=FALSE;
	bFileClose:=FALSE;
	bFilePuts:=FALSE;
	bFileGets:=FALSE;
END_IF

fbFileOpen(
	sNetId:='' ,
	sPathName:=sFileName ,
	nMode:=nOpenType ,
	ePath:=PATH_GENERIC ,
	bExecute:=bFileOpen ,
	tTimeout:=t#30s
);
hFileHandle:=fbFileOpen.hFile;
fbFileClose(
	sNetId:='' ,
	hFile:= hFileHandle ,
	bExecute:= bFileClose,
	tTimeout:= t#30s
);
fbFileGets(
	sNetId:= '' ,
	hFile:= hFileHandle ,
	bExecute:= bFileGets ,
	tTimeout:=t#30s
);
fbFilePuts(
	sNetId:= '',
	hFile:= hFileHandle,
	sLine:= ,
	bExecute:= bFilePuts ,
	tTimeout:= t#30s
);
END_PROGRAM

(* POU Programs/P_SaveData, ST *)
PROGRAM P_SaveData
VAR
	fbSaveData : FB_WritePersistentData;
	nMotorNominalRPMStore : UDINT := 0;
	sSerialNumberStore  : STRING(20) := '';		(* This holds the serial number of the machine *)
	sKaysJobNumberStore  : STRING(20) := '';		(* This holds the Kayse Engineering Job number of the machine *)
	sModelNumberStore : STRING(20) := '';		(* This variable holds the model of the machine *)
	sCustomerNameStore : STRING(20) := '';		(* This variable holds the customers name *)
	nMachineNumberStore : UDINT := 1;			(* The Machine Number designates what number the machines were delivered in for this series of special machines *)
	sProductionDateStore : STRING(10) := '';		(* This variable holds the date of production and should match that of the machine tags *)

	sLoadSideSetStore : STRING(30) :='None';	(* Holds the side that is currently set as Infeed *)
	nWAAxisThrustMaxStore: UDINT := 100;		(* Tailstock WA Axis Max Thrust *)
	nWBAxisThrustMaxStore: UDINT := 100;		(* Tailstock WB Axis Max Thrust *)
	nUAxisThrustMaxStore : UDINT :=100;		(* Max Thrust Set in secret screen *)
	fWAAxisHomeOffsetStore : LREAL;			(* A Tailstock WA Axis Offset Durring Homing *)
	fWBAxisHomeOffsetStore : LREAL;			(* B Tailstock WB Axis Offset Durring Homing *)
	fWAxisMoveOffBushingStore : LREAL;		(* Amount to Back W Axis' off of Bushing After Drill *)
	nTailstockClampingTorqueLimitStore: INT;
	fTailstockVelocityStore : LREAL;
	fUAxisVelocityStore : LREAL;
	fUAxisLoadSidePositionStore : LREAL;
	fUAxisUnloadSidePositionStore : LREAL;


	nCyclesCompleteStore : UDINT := 0;			(* Holds the # of completed cycles for Ream mode *)
	nMaxCyclesStore : UDINT := 0;				(* Holds the # of Max cycles for Ream mode *)
	sLastLoadedPartProgramNameStore : STRING(25) := '';
	fFlowMonitorMaxStore : LREAL := 0;
	bSideAEnabledStore : BOOL;					(* Enable of Machine Side B *)
	bSideBEnabledStore : BOOL;					(* Enable of Machine Side B *)


	(* Fault History Write Variables *)
	arrFaultHistoryStore : ARRAY[1..80] OF T_MaxString := 80('');	(* This holds the fault history array *)
	bFaultHistoryChanged : BOOL := FALSE;		(* bit to say that the stored value of Fault history does not match actual *)
	bFaultHistoryEmpty : BOOL := FALSE;			(* bit to say that the Fault history has not been loaded into the machine yet *)
	fbWriteFaultHistroyTrigger : TON;			(* A timer to delay the write of fault history *)
	nFaultHistoryStoreStep : UDINT := 0;			(* Fault History Write Counter *)
	nFaultHistoryReadStep : UDINT := 0;			(* Fault History Read Counter *)
	nReadLineStep : UDINT := 0;				(* Fault History Read Line Counter *)
	nCount: UDINT := 0;						(* Counter for Fault History Array *)
	nWriteLineStep : UDINT := 0;				(* Fault History Read Line Counter *)
	stFileName: T_MaxString := '';
	bFileClose: BOOL := FALSE;
	bFileWrite: BOOL := FALSE;
	bFileReadLine: BOOL := FALSE;
	bFileOpen: BOOL := FALSE;
	nOpenMode: UDINT := 0;
	fbFileOpen: FB_FileOpen;
	fbFileWrite: FB_FilePuts;
	fbFileReadLine: FB_FileGets;
	fbFileClose: FB_FileClose;
	nLoopIndex: UDINT := 0;						(* Counter for "FOR" loop  to Clear Fault History *)
	stOutVal: T_MaxString:='';					(* String to wrie to file *)
	stInVal: T_MaxString:='';					(* String to read from file *)

END_VAR
(* When one of the persistent data values change fromt he save value,
	then we trigger a write of the persistent data *)
IF 	nMotorNominalRPMStore<>nMotorNominalRPM OR
	sSerialNumberStore<>sSerialNumber OR
	sModelNumberStore<>sModelNumber OR
	sKaysJobNumberStore<>sKaysJobNumber OR
	sCustomerNameStore<>sCustomerName OR
	sProductionDateStore<>sProductionDate OR
	nMachineNumberStore <> nMachineNumber OR
	nCyclesCompleteStore<>nCyclesComplete OR
	nMaxCyclesStore<>nMaxCycles OR
	sLastLoadedPartProgramNameStore<>sLastLoadedPartProgramName OR
	fFlowMonitorMaxStore<>fFlowMonitorMax OR

	sLoadSideSetStore <> sLoadSideSet OR
	nUAxisThrustMaxStore <> nUAxisThrustMax OR
	fWAAxisHomeOffsetStore <> fWAAxisHomeOffset OR
	fWBAxisHomeOffsetStore <> fWBAxisHomeOffset OR
	fWAxisMoveOffBushingStore <> fWAxisMoveOffBushing OR
	nTailstockClampingTorqueLimitStore <> nTailstockClampingTorqueLimit OR
	fTailstockVelocityStore <> fTailstockVelocity OR
	bSideAEnabledStore <> bSideAEnabled OR
	bSideBEnabledStore <> bSideBEnabled OR
	fUAxisVelocityStore <> fUAxisVelocity OR
	fUAxisLoadSidePositionStore <> fUAxisLoadSidePosition OR
	fUAxisUnloadSidePositionStore <> fUAxisUnloadSidePosition

THEN
	fbSaveData(
		NETID:= ,
		PORT:=801 ,
		START:=TRUE ,
		TMOUT:=t#5s ,
		MODE:=SPDM_2PASS ,
		BUSY=> ,
		ERR=> ,
		ERRID=> );
	IF NOT(fbSaveData.BUSY) THEN
		nMotorNominalRPMStore:=nMotorNominalRPM;
		sSerialNumberStore:= sSerialNumber;
		sModelNumberStore:= sModelNumber;
		sKaysJobNumberStore:= sKaysJobNumber;
		sCustomerNameStore:= sCustomerName;
		sProductionDateStore:= sProductionDate;
		nMachineNumberStore := nMachineNumber;
		nCyclesCompleteStore := nCyclesComplete;
		nMaxCyclesStore := nMaxCycles;
		sLastLoadedPartProgramNameStore := sLastLoadedPartProgramName;
		fFlowMonitorMaxStore := fFlowMonitorMax;

		sLoadSideSetStore := sLoadSideSet;
		nUAxisThrustMaxStore := nUAxisThrustMax;
		fWAAxisHomeOffsetStore := fWAAxisHomeOffset;
		fWBAxisHomeOffsetStore := fWBAxisHomeOffset;
		fWAxisMoveOffBushingStore := fWAxisMoveOffBushing;
		nTailstockClampingTorqueLimitStore := nTailstockClampingTorqueLimit;
		fTailstockVelocityStore := fTailstockVelocity;
		bSideAEnabledStore := bSideAEnabled;
		bSideBEnabledStore := bSideBEnabled;
		fUAxisLoadSidePositionStore := fUAxisLoadSidePosition;
		fUAxisUnloadSidePositionStore := fUAxisUnloadSidePosition;
		fUAxisVelocityStore := fUAxisVelocity;

	END_IF
ELSE
	fbSaveData(START:=FALSE);
END_IF

(*		FAULT HISTORY Save 		*)
(*
IF MEMCMP(ADR(arrFaultHistory), ADR(arrFaultHistoryStore), SIZEOF(arrFaultHistory))<>0 THEN
	bFaultHistoryChanged:=TRUE;
ELSE (* Once they match then turn off bit *)
	bFaultHistoryChanged:=FALSE;
END_IF

(* Wait 1.5 minute after the fault history has changed to store to disk *)
fbWriteFaultHistroyTrigger(in:=bFaultHistoryChanged, PT:=t#90s);

(* Set a Trigger on first Scan to say the Fault History needs to be loaded from file *)
IF SystemTaskInfoArr[1].firstCycle THEN
	bFaultHistoryEmpty:=TRUE;
END_IF

(* Give Reading Priority by position, and do not read and write at the same time *)
IF bFaultHistoryEmpty THEN
	CASE nFaultHistoryReadStep OF
	0: (* Setup *)
		sFileOpError:='';
		(* Prepare For Next Step *)
		nOpenMode:=FOPEN_MODEREAD OR FOPEN_MODETEXT;
		bFileOpen:=FALSE;
		(* Move To Next Step *)
		nFaultHistoryReadStep:=nFaultHistoryReadStep+1;

	1: (* Open The File *)

		(* Check For Completion Of Operation *)
		IF NOT(fbFileOpen.bBusy) AND NOT(fbFileOpen.bError) AND bFileOpen THEN
			(* Prepare For Next Step *)
			bFileReadLine:=FALSE;
			nReadLineStep:=0;
			nCount:=1;
			bFileOpen:=FALSE;
			(* Move To Next Step *)
			nFaultHistoryReadStep:=nFaultHistoryReadStep+1;
		(* Check For Error Condition *)
		ELSIF fbFileOpen.bError AND bFileOpen THEN
			sFileOpError:=CONCAT('Fault History Read Open Error:  ',UDINT_TO_STRING(fbFileOpen.nErrId));
			bFileOpen:=FALSE;
			nFaultHistoryReadStep:=70;
		ELSE
			bFileOpen:=TRUE;
		END_IF

	2: (* Read The File - line by line *)

		CASE nReadLineStep OF
		0: (* Wait For Read To Finish *)
			IF NOT(fbFileReadLine.bBusy) AND bFileReadLine THEN
				(* Toggle off Trigger *)
				bFileReadLine:=FALSE;
				nReadLineStep:=nReadLineStep+1;
			ELSE (* Get The Next Line Of The File *)
				bFileReadLine:=TRUE;
			END_IF

		1: (* Store Retrieved String *)
			stInVal:=fbFileReadLine.sLine;
			(* Move To Next Step *)
			nReadLineStep:=nReadLineStep+1;

		2: (* Check for Read error or End Of File - There should only be 80 lines max  *)
			IF fbFileReadLine.bEOF OR nCount>80 THEN
				(* Move Out of Reading line *)
				nFaultHistoryReadStep:=nFaultHistoryReadStep+1;
				(* Prepare For Next Step *)
				bFileClose:=FALSE;
			ELSIF fbFileReadLine.bError THEN
				(* Error Report And Close File *)
				sFileOpError:=CONCAT('Fault History Read Line Error:  ',UDINT_TO_STRING(fbFileReadLine.nErrId));
				bFileClose:=FALSE;
				nFaultHistoryReadStep:=70;
			ELSE (* Move To Next Step *)
				nReadLineStep:=nReadLineStep+1;
			END_IF

		3: (* Write the value to Array Fault History *)
			(* Extract the End of line character and put the string into the Array *)
			arrFaultHistory[nCount]:=DELETE(stInVal,1,LEN(stInVal));
			(* Jump back to read next line *)
			nCount:=nCount+1;
			bFileReadLine:=FALSE;
			nReadLineStep:=0;

		END_CASE

	3: (*Close file *)
		(* Check For Completion *)
		IF NOT( fbFileClose.bBusy) AND bFileClose THEN
			bFileClose:=FALSE;
			(* Move To Next Step *)
			nFaultHistoryReadStep:=nFaultHistoryReadStep+1;
		(* Check For Error Condition *)
		ELSIF fbFileClose.bError THEN
			sFileOpError:=CONCAT('Fault History Read Close Error:  ',UDINT_TO_STRING(fbFileClose.nErrId));
			bFileClose:=FALSE;
			nFaultHistoryReadStep:=70;
		ELSE
			bFileClose:=TRUE;
		END_IF

	4: (* Done *)
		bFaultHistoryEmpty:=FALSE;
		nFaultHistoryReadStep:=0;

	70: (* Error Recovery *)
		bFaultHistoryEmpty:=FALSE;
		bFaultHistoryFileError:=TRUE;
		nFaultHistoryReadStep:=0;

	END_CASE


ELSIF fbWriteFaultHistroyTrigger.Q THEN

	CASE nFaultHistoryStoreStep OF
	0: (* Setup *)
		sFileOpError:='';
		(* Prepare For Next Step *)
		nOpenMode:=FOPEN_MODEWRITE OR FOPEN_MODETEXT;
		bFileOpen:=FALSE;
		(* Move To Next Step *)
		nFaultHistoryStoreStep:=nFaultHistoryStoreStep+1;

	1: (* Open/Create The File *)
		(* Check For Completion *)
		IF NOT(fbFileOpen.bBusy) AND NOT(fbFileOpen.bError) AND bFileOpen THEN
			bFileOpen:=FALSE;
			bFileWrite:=FALSE;
			nCount:=1;
			nWriteLineStep:=0;
			stOutVal:='';
			nFaultHistoryStoreStep:=nFaultHistoryStoreStep+1;
		(* Check For Error Condition *)
		ELSIF fbFileOpen.bError AND bFileOpen THEN
			sFileOpError:=CONCAT('Fault History Write Open Error:  ',UDINT_TO_STRING(fbFileOpen.nErrId));
			bFileOpen:=FALSE;
			nFaultHistoryStoreStep:=70;
		(*Trigger a file Open to Create/empty the file *)
		ELSE
			bFileOpen:=TRUE;
		END_IF

	2: (* Write file to disk Line by Line *)
		CASE nWriteLineStep OF
			0: (* Create String to write *)
				(* Done if Fault History Array element is blank or above 80 lines *)
				IF arrFaultHistory[nCount]='' OR nCount>=80 THEN
					bFileWrite:=FALSE;
					bFileClose:=FALSE;
					nFaultHistoryStoreStep:=nFaultHistoryStoreStep+1;
				(* Write sting and add EOL character *)
				ELSE
					stOutVal:=arrFaultHistory[nCount];
					stOutVal:=CONCAT(stOutVal,'$L');
					(* Prepare For Next Step *)
					fbFileWrite.sLine:=stOutVal;
					bFileWrite:=FALSE;
					nWriteLineStep:=nWriteLineStep+1;
				END_IF

			1: (* Write Line to Disk *)
				(* Check For Completion *)
				IF NOT( fbFileWrite.bBusy) AND NOT(fbFileWrite.bError) AND bFileWrite THEN
					(* Incriment count for next line *)
					nCount:=nCount+1;
					stOutVal:='';
					(* Jump back to create next line *)
					bFileWrite:=FALSE;
					nWriteLineStep:=0;
				(* Check For Error Condition *)
				ELSIF fbFileWrite.bError AND bFileWrite THEN
					sFileOpError:=CONCAT('Fault History Write Error:  ',UDINT_TO_STRING(fbFileWrite.nErrId));
					bFileWrite:=FALSE;
					bFileClose:=TRUE;
					nFaultHistoryStoreStep:=70;
				ELSE (* Initiate write *)
					bFileWrite:=TRUE;
				END_IF
		END_CASE
	3: (*Close the File *)
		(* Check For Completion *)
		IF NOT( fbFileClose.bBusy) AND NOT(fbFileClose.bError) AND bFileClose THEN
			(* Move To Next Step *)
			nFaultHistoryStoreStep:=nFaultHistoryStoreStep+1;
			bFileClose:=FALSE;
		(* Check For Error Condition *)
		ELSIF fbFileClose.bError AND bFileClose THEN
			sFileOpError:=CONCAT('Fault History Close Error:  ',UDINT_TO_STRING(fbFileClose.nErrId));
			nFaultHistoryStoreStep:=70;
		ELSE
			bFileClose:=TRUE;
		END_IF

	4: (* Set the Array Store Value to ArrayFaultHistory *)
		MEMCPY(ADR(arrFaultHistoryStore), ADR(arrFaultHistory), SIZEOF(arrFaultHistory));
		(* This will automatically turn off bFaultHistoryChanged, so fbWriteFaultHistroyTrigger.Q will go off *)
		nFaultHistoryStoreStep:=0;

	70: (* Error State *)
		bFaultHistoryFileError:=TRUE;
		bFileClose:=FALSE;
		bFaultHistoryChanged:=FALSE; (* turn off the condition for the elsif of this case *)
		nFaultHistoryStoreStep:=0;

	END_CASE
(* Clear the 80 lines of FAult History *)
ELSIF bClearFAultHistoryPB THEN
	FOR nLoopIndex:=1 TO 80 BY 1 DO
		arrFaultHistory[nLoopIndex]:='';
	END_FOR;
	IF nLoopIndex>=80 THEN
		bClearFAultHistoryPB:=FALSE;
	END_IF
END_IF
*)

fbFileOpen(
	sNetId:='' ,
	sPathName:='\Hard Disk\ftp\FaultHistory.csv' ,
	nMode:= nOpenMode,
	ePath:=PATH_GENERIC ,
	bExecute:=bFileOpen ,
	tTimeout:=t#10s );
fbFileReadLine(
	sNetId:='' ,
	hFile:=fbFileOpen.hFile ,
	bExecute:=bFileReadLine ,
	tTimeout:=t#10s,
	bBusy=> ,
	bError=> ,
	nErrId=> ,
	sLine=> ,
	bEOF=> );
fbFileWrite(
	sNetId:='' ,
	hFile:=fbFileOpen.hFile ,
	sline:=stOutVal ,
	bExecute:=bFileWrite ,
	tTimeout:=t#10s );
fbFileClose(
	sNetId:='' ,
	hFile:=fbFileOpen.hFile ,
	bExecute:=bFileClose ,
	tTimeout:=t#10s );
END_PROGRAM

(* POU Programs/P_TransferControl, ST *)
PROGRAM P_TransferControl
VAR
	bTransferAxisEnable: BOOL;
	fbTransferAxisPower: MC_Power;
	fbTransferAxisMove: MC_MoveAbsolute;
	fbTransferAxisSetZero: MC_SetPosition;
	fbTransferAxisStop: MC_Stop;
	bTransferAxisPower: BOOL := FALSE;
	bTransferAxisHome: BOOL := FALSE;
	bTransferAxisMove: BOOL := FALSE;
	fTransferMovePosition : LREAL := 0.0;
	bTransferAxisStop: BOOL := FALSE;
	bTransferAxisSetZero: BOOL := FALSE;
	fTransferAxisSetZeroPosition: LREAL := 0.0;
	fbHomeUPBRTrig: R_TRIG;				(* Capture the Rising edge of the Home PB *)

	bManualLower: BOOL := FALSE;				(*Manual Set Lower Carrier Cylinder*)
	bManualRaise: BOOL := FALSE;				(*Manual Set Raise Carrier Cylinder*)

(* Inputs *)
	(* bEnable *)
	bSideADisabled : BOOL := FALSE;		(* Set by Supervisory Personnell if Side A is to be disabled *)
	bSideBDisabled : BOOL := FALSE;		(* Set by Supervisory Personnell if Side A is to be disabled *)
	(* PartLoadCompletePB *)				(* Operator Pendant Push Button *)
	(* All of the Load and Unload Nest Proxes should be inputs *)
	(* Raise and Lower Transfer Proxes should be inputs *)
	bSideAClampComplete: BOOL := FALSE;			(* Signal from the Tailstock that it has clamped the parts - OK to lower *)
	bSideBClampComplete: BOOL := FALSE;			(* Signal from the Tailstock that it has clamped the parts - OK to lower *)

(*Outputs *)
	bSideAReadyToClamp : BOOL := FALSE;	(* Output to Tailstock to say Side A is ready to clamp Parts *)
	bSideBReadyToClamp : BOOL := FALSE;	(* Output to Tailstock to say Side B ready to clamp Parts *)

(* Cycle Variables *)

	fbMoveToUnloadRTrig: R_TRIG;
	bAutoMoveToDrill: BOOL := FALSE;
	fbDownAndLoadRTrig: R_TRIG;
	fbAutoTransferWatchdog : TON;
	bAutoTransferWatchdog : BOOL := FALSE;
	tAutoTransferWatchdogTime : TIME;
	fbUAxisStopTrig: R_TRIG;		(* Trigger a Stop of the Transfer U Axis*)
	fbCellRunoutTrig: R_TRIG;		(* R_Trig of the Cell Runout PB was pressed *)
	bLoadSideClearOfParts: BOOL := FALSE;		(* The Load Side does not have any parts loaded*)

	fbTransferUpOffDelay: TON;			(* Delay time of the Raise Output being Off *)
	fbTransferDownOffDelay: TON;			(* Off Delay time of the Lower Output being Off *)

	bTransferEnabled: BOOL := FALSE;		(* Transfer Enable Signal *)
	nTransferState: UDINT := 0;				(* Transfer State Case/Counter Variable *)
	nTransferAutoStep: UDINT := 0;			(* Transfer Automatic Step Case/Counter Variable *)
	nTransferManualStep: UDINT := 0;		(* Transfer Manual Step Case/Counter Variable *)
	bUDeCtrlEnable: BOOL := FALSE;		(* Enable Bit for FB to Move off Overtravel *)
END_VAR
(*Call the Action Transfer Cycle *)
Transfer_Cycle;

(* When we are in Manual Mode we do not need to display message waiting on Unload Confirm *)
IF NOT(bMachineMode) THEN
	bDisplayUnloadConf:=FALSE;
END_IF

(* We need to know when the load and Unload sides are clear of parts *)
IF (sLoadSideSet = 'A') THEN
	bUnloadSideClearOfParts := NOT(bProx510 OR bProx511 OR bProx512 OR bProx513 OR bProx514 OR bProx515);
	bLoadSideClearOfParts := NOT( bProx410 OR bProx411 OR bProx412 OR bProx413 OR bProx414 OR bProx415);
ELSIF (sLoadSideSet ='B') THEN
	bUnloadSideClearOfParts := NOT( bProx410 OR bProx411 OR bProx412 OR bProx413 OR bProx414 OR bProx415);
	bLoadSideClearOfParts := NOT(bProx510 OR bProx511 OR bProx512 OR bProx513 OR bProx514 OR bProx515);
END_IF

(* When the Transfer Down and Load signal is on we want to turn it off when the transfer gets back to the Load postion and is down.
	We cant do this in the Drill Cycle because the transfer movements are somewhat independant of the drill cycle. *)
IF bAutoTransferDownAndLoad AND bProx517 AND bTransferAtLoadIndicator THEN
	bAutoTransferDownAndLoad:=FALSE;
END_IF

(* Turn on the Power to Transfer Axis when Hard Enable is on *)
bTransferAxisPower := bUServoEnable;

fbTransferAxisPower(
	Enable:=bTransferAxisPower ,
	Enable_Positive:=bTransferAxisPower ,
	Enable_Negative:=bTransferAxisPower ,
	Override:=100 ,
	BufferMode:=MC_Aborting ,
	Axis:=stUAxis );

(* When the Stop is Done or has an error then we turn off the trigger *)
IF fbUAxisStop.Done OR fbUAxisStop.Error THEN
	bUStop:=FALSE;
END_IF
fbUAxisStop(
	Execute := bUStop,
	Deceleration := 0,
	Jerk := 0,
	Axis := stUAxis );

fbTransferAxisMove(
	Execute:= bTransferAxisMove ,
	Position:= fTransferMovePosition ,
	Velocity:= fTransferMoveVelo ,
	Acceleration:= 0 ,
	Deceleration:= 0,
	Jerk := 0,
	BufferMode:=MC_Aborting ,
	Axis := stUAxis );

fbUAxisMCReset(
	Execute:=bUMCResetRequest ,
	Axis:=stUAxis );

fbUAxisDriveReset(
	NetId:='' ,
	Execute:=bUDriveResetRequest ,
	Timeout:=t#10s ,
	Axis:= stUAxis, );

stUAxis.ReadStatus();

(* If one of the U Axis overtravel limit switches is made, then turn on the bit that allows
Movement off of the limit switchs 
NOTE: The U Axis uses Prox sensors instead of NC Limit Switches so the next line is different *)
IF (DriveUdinputs.0) OR (DriveUdinputs.1) THEN
	bUDeCtrlEnable:=TRUE;
ELSE
	bUDeCtrlEnable:=FALSE;
END_IF
stUAxis.PlcToNc.ControlDWord :=
AxisSetAcceptBlockedDriveSignal(stUAxis.PlcToNc.ControlDWord,
	bEnable:= bUDeCtrlEnable );

(* If a Drive reset was requested then when the Drive Reset is done we want to do a MC Reset of the NC Axis *)
IF bUDriveResetRequest AND (NOT (fbUAxisDriveReset.Busy) OR  fbUAxisDriveReset.Error) THEN
	bUMCResetRequest:=TRUE;
END_IF
IF fbUAxisMCReset.Done OR fbUAxisMCReset.Error THEN
	buMCResetRequest:=FALSE;
	bUDriveResetRequest:=FALSE;
END_IF

(* When the Home PB pressed trigger a home *)
fbHomeUPBRTrig(CLK:=bHomeUAxisPB);
IF fbHomeUPBRTrig.Q THEN
	bUAxisHome:=TRUE;
(* When Home is done turn off trigger *)
ELSIF fbTransferAxisHome.Done THEN
	bUAxisHome:=FALSE;
(* If an Error Occurs then turn off trigger and Issue a Stop command *)
ELSIF  fbTransferAxisHome.Error  THEN
	bUAxisHome:=FALSE;
	bUStop:=TRUE;
END_IF

fbTransferAxisHome(
	Execute:= bUAxisHome ,
	Position:=0 ,
	HomingMode:= ,
	BufferMode:= ,
	Options:= ,
	bCalibrationCam:= DriveUdinputs.5 ,
	Axis:= stUAxis ,
	Done=> ,
	Busy=> ,
	Active=> ,
	CommandAborted=> ,
	Error=> ,
	ErrorID=>  );

(* 	SOLENOID VALVE CONTROL 	*)
(* This part of the programs handles the solenoid valves for the raising and lowering of the Transfer.
	It prohibits Solenoid A and B being fired at the same time and when the hydraulic unit is running and
	Manual mode is entered it fires the solenoid that corresponds to the feedback inputs *)

(* Fire Solenoid Valves *)
(* Must have MCR and Hydraulic Unit *)
IF bMCR AND bHydraulicPowerUnitRunning
	(* When Drill Return Activated we want to turn off the outputs to stop motion *)
	AND ( NOT nActiveFaults[1].1 AND bPB4ADrillReturn AND bPB4BDrillReturn )
THEN
	IF NOT(bMachineMode) AND bManualRaise OR
		bMachineMode AND bAutoRaise
	THEN
		bTransferDown := FALSE;
		IF fbTransferDownOffDelay.Q THEN
			bTransferUp := TRUE;
		END_IF
	ELSIF NOT(bMachineMode) AND bManualLower OR
		bMachineMode AND bAutoLower
	THEN
		bTransferUp := FALSE;
		IF fbTransferDownOffDelay.Q THEN
			bTransferDown := TRUE;
		END_IF
	END_IF
(* When the MCR is off or Hydraulics Off, we turn off the solenoids *)
ELSE (* NOT Enabled *)
	bTransferDown:=FALSE;
	bTransferUp:=FALSE;
END_IF

(* These timers help not to turn on the opposing solenoid until we make sure the coil is fully de-enrgized *)
fbTransferUpOffDelay(IN:=NOT bTransferUp, PT:= t#100ms);
fbTransferDownOffDelay(IN:= NOT bTransferDown, PT:= t#100ms);

(*FAIL-SAFE CONTROL
If Both Outputs are on at the same time then turn them Off and Fault *)
IF bTransferDown AND bTransferUp THEN
	nModeError:=Er_TransferSolError;
	bTransferDown:=FALSE;
	bTransferUp:=FALSE;
END_IF
END_PROGRAM
ACTION Transfer_Cycle:
(* This part handles the action of moving the Transfer from the Load to Unload position
     and Lowering the transfer and moving it to the Load position.  Each is triggered by the Auto cycle *)

bTransferEnabled:= bMCC_SConfirm AND bHydraulicPowerUnitRunning;


(* Confirm Enable is active - if not then Clear all states *)
IF bTransferEnabled THEN
	(*Transfer Current States:
		0= Decide if in Manual or Auto
		1= Manual Mode
		2= Auto Mode
		255= Error State	*)
	CASE nTransferState OF
	0:(* Initialize - Select between Auto or Manual *)
		(* Manual and Auto Mode are Mutually Exclusive inputs *)
		IF NOT(bMachineMode) THEN (* Manual Mode *)
			nTransferState:=1;
			nTransferAutoStep:=0;
		ELSE	(* Auto Mode *)
			nTransferState:=2;
			nTransferManualStep:=0;
		END_IF

	1: (*** MANUAL MODE ***)
		CASE nTransferManualStep OF
		0: (* Initial State *)
			(* Turn off all Auto Signals signals *)
			bAutoRaise := FALSE;
			bAutoLower := FALSE;
			bAutoTransferWatchdog:=FALSE;
			bCellRunoutRequest:= FALSE;
			bDispPressCycleStart:=FALSE;
			bLoadPartsConfirmed:= FALSE;
			bAutoTransferPartsToDrill:=FALSE;
			bAutoTransferDownAndLoad:=FALSE;
			nTransferAutoStep:=0;
			nTransferManualStep:=nTransferManualStep+1;

		1: (* This Step Checks Sensor Inputs to determine what Solenoids should be fired *)
			(* Only evaluate when no fault or Drill Return *)
			IF NOT bMachineFault AND bPB4ADrillReturn AND bPB4BDrillReturn THEN
				(*** TRANSFER RAISE/LOWER CYLINDER ***)
				(* Lower  if Prox is confirming position *)
				IF bProx517 THEN
					bManualLower := TRUE;
					bManualRaise := FALSE;
				(* Raise if Prox is confirming position  *)
				ELSIF bProx516 THEN
					bManualLower := FALSE;
					bManualRaise :=TRUE;
				(* No Sensor Confirmation - Unknown State - Turn Both Off *)
				ELSE
					bManualLower := FALSE;
					bManualRaise := FALSE;
				END_IF
			(* If Fault we want to turn off the Manual Raise & Lower Outputs to hold position *)
			ELSE	bManualLower := FALSE;
					bManualRaise := FALSE;
			END_IF
			nTransferManualStep:=nTransferManualStep+1;

		(* Always Return to this Step while in manual *)
		2: (* Evaluate What To Do Next *)

			(* If We have a fault do not allow manual functions *)
			IF bMachineFault THEN
				bTransferAxisMove := FALSE;
				bManualLower := FALSE;
				bManualRaise := FALSE;
			(* Leaving Manual Mode *)
			ELSIF bMachineMode THEN
				bManualLower := FALSE;
				bManualRaise := FALSE;
				nTransferManualStep:=0;
				nTransferState:=0;
			(* Push Buttons - Axis Must Not be Moving *)
			ELSIF bTransferDownPB AND NOT(fbTransferAxisMove.Busy) THEN
				bManualLower := TRUE;(* probar cambio a False que hace *)
				bManualRaise := FALSE;
			ELSIF bTransfer
PB AND NOT(fbTransferAxisMove.Busy) THEN
				bManualLower := FALSE;
				bManualRaise :=TRUE;(* probar cambio a False que hace *)
			(* W and U Axis Homed *)
			(* When the PB's are pressed then initiate the Move
				the PB's are pulsed from the panel side. *)
			ELSIF bMoveUtoLoadPB AND NOT(fbTransferAxisMove.Busy) THEN
				IF bWandUAxisHomed THEN
					bTransferAxisMove := TRUE;(* probar cambio a False que hace *)
					fTransferMovePosition := fUAxisLoadSidePosition;
				ELSE (* W and U axis NOT homed *)
					bTransferError := TRUE;
					nTransferErrorID := 7;
					nTransferState := 255;
				END_IF
			ELSIF bMoveUtoUnloadPB AND NOT(fbTransferAxisMove.Busy) THEN
				IF bWandUAxisHomed THEN
					bTransferAxisMove := TRUE;
					fTransferMovePosition := fUAxisUnloadSidePosition;
				ELSE (* W and U axis NOT homed *)
					bTransferError := TRUE;
					nTransferErrorID := 7;
					nTransferState := 255;
				END_IF
			ELSE
				bTransferAxisMove := FALSE;
			END_IF

		END_CASE	(* nTransferManualStep *)

	2: (*** AUTO MODE ***)
		nTransferManualStep:=0;

		(* If we leave Auto turn off any outputs that are causing motion.
		 When Manual is entered it will check the state and turn on the appropriate outputs based upon sensor states 
		 Also we want to issue a stop command to the transfer *)
		IF NOT(bMachineMode) THEN (* Manual Mode *)
			(* Turn off Rais and Lower signals *)
			bAutoRaise := FALSE;
			bAutoLower := FALSE;
			bAutoTransferWatchdog:=FALSE;
			bCellRunoutRequest:= FALSE;
			bLoadPartsConfirmed:= FALSE;
			bAutoTransferPartsToDrill:=FALSE;
			bAutoTransferDownAndLoad:=FALSE;
			nTransferAutoStep:=0;
			(* Stop the Axis *)
			IF bTransferAxisMove THEN
				bTransferAxisMove := FALSE;
				nTransferState:=254;
			ELSE
				nTransferState:=0;
			END_IF
		END_IF

		(* Safety interlock: while drilling/retracting keep transfer idle and stop active U-axis moves. *)
		IF nAutoCycleStep=AC_Drill
			OR nAutoCycleStep=AC_DrillReturn
			OR nAutoCycleStep=AC_Retract
		THEN
			bAutoTransferPartsToDrill:=FALSE;
			bAutoTransferDownAndLoad:=FALSE;
			bAutoRaise:=FALSE;
			bAutoLower:=FALSE;
			bAutoTransferWatchdog:=FALSE;
			nTransferAutoStep:=2;
			IF bTransferAxisMove THEN
				bTransferAxisMove:=FALSE;
				nTransferState:=254;
			END_IF
		END_IF

		CASE nTransferAutoStep OF
		0: (* Initial Step *)
			bAutoTransferWatchdog:=FALSE;
			nTransferAutoStep:=nTransferAutoStep+1;

		1: (* Check state of the transfer *)
			(* These conditions will Fault so we will Exit Auto *)

			(* We want to be Down and at the Load Position *)
			(* Fault - Both Up and Down proxes on at same time *)
			IF bProx516 AND bProx517 THEN
				bTransferError := TRUE;
				nTransferErrorID := 54;
				nTransferState := 255;
			(* Fault - Not Down *)
			ELSIF bProx516 OR NOT(bProx517) THEN
				bTransferError := TRUE;
				nTransferErrorID := 52;
				nTransferState := 255;
			(* Fault - Not Homed *)
			ELSIF NOT bWandUAxisHomed THEN
				bTransferError := TRUE;
				nTransferErrorID := 53;
				nTransferState := 255;
			(* Fault - Actual position not within +/- 0.5mm of Load Position *)
			ELSIF NOT bTransferAtLoadIndicator THEN
				bTransferError := TRUE;
				nTransferErrorID := 50;
				nTransferState := 255;
			(* Conditions are good for enteing Auto *)
			ELSE
				nTransferAutoStep:=nTransferAutoStep+1;
			END_IF

		2: (* Always Return to Here to wait for next command *)
			(* Leaving Auto is handled above *)
			(* Must be In Cycle to trigger these Automatic functions *)
			IF bInCycle THEN
				(* Cell Runout Activation *)
				IF fbCellRunoutTrig.Q THEN
					 (* Set number of transfer cycles required before turning off request *)
					IF bLoadPartsConfirmed THEN
						nCellRunoutCounter:=3;
					ELSE
						nCellRunoutCounter:=2;
					END_IF
					bCellRunoutRequest:= TRUE;
				END_IF

				(* Decide what Automatic Function to do *)
				(* Raise the Transfer - Parts Loaded *)
				IF bLoadPartsConfirmed AND bTransferAtLoadIndicator AND bProx517 THEN
					bLoadPartsConfirmed:= FALSE;
					nTransferAutoStep:=10;
				(* Move Transfer to Drill/Unload *)
				ELSIF fbProx516TON.Q AND  bAutoTransferPartsToDrill THEN
					nTransferAutoStep:=30;
				(* Raise the Transfer - Cell Runout *)
				ELSIF bCellRunoutRequest  AND bTransferAtLoadIndicator THEN
					nTransferAutoStep:=15;
				(* Lower Transfer and Move to Load Postion triggered *)
				ELSIF fbDownAndLoadRTrig.Q THEN
					nTransferAutoStep:=40;
				END_IF
			ELSE
				bCellRunoutRequest:= FALSE;
				nCellRunoutCounter:=0;
				bLoadPartsConfirmed:= FALSE;
				bAutoTransferPartsToDrill:=FALSE;
				bAutoTransferDownAndLoad:=FALSE;
			END_IF


		10:(* Check for Parts Load Side *)
			(* Load side set to A *)
			IF  sLoadSideSet = 'A' THEN
				(* When A side not enabled there should be no parts *)
				IF NOT(bSideAEnabled)  AND (bProx410 OR bProx411 OR bProx412) THEN
					bLoadPartsConfirmed := FALSE;
					bTransferError := TRUE;
					nTransferErrorID := 11;
					nTransferState := 255;
				(* When A side enabled all parts should be there *)
				ELSIF bSideAEnabled AND (NOT bProx410 OR NOT bProx411 OR NOT bProx412) THEN
					bLoadPartsConfirmed := FALSE;
					bTransferError := TRUE;
					nTransferErrorID := 12;
					nTransferState := 255;
				(* When Side B not enabled there should be no parts *)
				ELSIF NOT(bSideBEnabled) AND (bProx413 OR bProx414 OR bProx415) THEN
					bLoadPartsConfirmed := FALSE;
					bTransferError := TRUE;
					nTransferErrorID := 13;
					nTransferState := 255;
				(* When B side enabled all parts should be there *)
				ELSIF bSideBEnabled AND (NOT bProx413 OR NOT bProx414 OR NOT bProx415) THEN
					bLoadPartsConfirmed := FALSE;
					bTransferError := TRUE;
					nTransferErrorID := 14;
					nTransferState := 255;
				(* Passed checks so raise transfer *)
				ELSE
					IF bCellRunoutRequest THEN
						bLoadPartsConfirmed := FALSE;
						nTransferAutoStep:=15;
					ELSE
						bLoadPartsConfirmed := FALSE;
						nTransferAutoStep:=20;
					END_IF
				END_IF
			(* Load side set to B *)
			ELSIF sLoadSideSet ='B' THEN
				(* When A side not enabled there should be no parts *)
				IF NOT(bSideAEnabled) AND (bProx510 OR bProx511 OR bProx512) THEN
					bLoadPartsConfirmed := FALSE;
					bTransferError := TRUE;
					nTransferErrorID := 11;
					nTransferState := 255;
				(* When A side enabled all parts should be there *)
				ELSIF bSideAEnabled AND (NOT bProx510 OR NOT  bProx511 OR NOT bProx512) THEN
					bLoadPartsConfirmed := FALSE;
					bTransferError := TRUE;
					nTransferErrorID := 12;
					nTransferState := 255;
				(* When Side B not enabled there should be no parts *)
				ELSIF NOT(bSideBEnabled) AND (bProx513 OR bProx514 OR bProx515) THEN
					bLoadPartsConfirmed := FALSE;
					bTransferError := TRUE;
					nTransferErrorID := 13;
					nTransferState := 255;
				(* When B side enabled all parts should be there *)
				ELSIF bSideBEnabled AND (NOT bProx513 OR NOT bProx514 OR NOT bProx515) THEN
					bLoadPartsConfirmed := FALSE;
					bTransferError := TRUE;
					nTransferErrorID := 14;
					nTransferState := 255;
				(* Passed checks so raise transfer *)
				ELSE
					IF bCellRunoutRequest THEN
						bLoadPartsConfirmed := FALSE;
						nTransferAutoStep:=15;
					ELSE
						bLoadPartsConfirmed := FALSE;
						nTransferAutoStep:=20;
					END_IF
				END_IF
			END_IF

		15: (* Make Sure there are no parts on Load Side for Cell Runout *)
			IF  bLoadSideClearOfParts THEN
				nTransferAutoStep:=20;
			ELSE
				IF bTransferError THEN
					nTransferState := 255;
				END_IF
				bTransferError := TRUE;
				nTransferErrorID := 1;
			END_IF

		(* Raise Transfer *)
		20: (* Check Transfer Position and Down *)
			bAutoLower := FALSE;
			IF NOT bTransferAtLoadIndicator THEN
				bTransferError := TRUE;
				nTransferErrorID := 16;
				nTransferState := 255;
			ELSE
				bAutoRaise := TRUE;
				bAutoTransferWatchdog:=TRUE;
				tAutoTransferWatchdogTime := t#20s;
				nTransferAutoStep:=21;
			END_IF

		21: (* Wait for Transfer Raise *)
			(* Fault - Raise took to long *)
			IF fbAutoTransferWatchdog.Q THEN
				bAutoTransferWatchdog:=FALSE;
				bAutoRaise := FALSE;
				bTransferError := TRUE;
				nTransferErrorID := 2;
				nTransferState := 255;
			(* Fault - Both Up and Down Proxes on *)
			ELSIF bProx517 AND bProx516 THEN
				bAutoTransferWatchdog:=FALSE;
				bAutoRaise := FALSE;
				bTransferError := TRUE;
				nTransferErrorID := 3;
				nTransferState := 255;
			(* Done with Raise *)
			ELSIF fbProx516TON.Q AND bAutoRaise THEN
				bAutoTransferWatchdog:=FALSE;
				nTransferAutoStep:=22;
			END_IF

		22: (* Check Load Side Proxes are all  Off *)
			IF bLoadSideClearOfParts THEN
				nTransferAutoStep:=2;
			ELSE
				bTransferError := TRUE;
				nTransferErrorID := 8;
				nTransferState := 255;
			END_IF


		(* Transfer to Drill/Unload *)
		30: (* Check for Parts on Unload Side and Transfer UP *)
			bLoadPartsConfirmed := FALSE;
			IF NOT  bUnloadSideClearOfParts THEN
				bTransferError := TRUE;
				nTransferErrorID := 17;
				nTransferState := 255;
			(* Check Transfer Up *)
			ELSIF NOT(fbProx516TON.Q) AND bProx517 THEN
				bTransferError := TRUE;
				nTransferErrorID := 9;
				nTransferState := 255;
			(* Checks OK *)
			ELSE
				nTransferAutoStep:=31;
			END_IF

		31: (* Check W Axis Positions *)
			(* When A enabled WA must be back *)
			IF bSideAEnabled AND NOT( (fWAxisTransferPosition-0.2) <= stWAAxis.NcToPlc.ActPos ) THEN
				bAutoTransferPartsToDrill := FALSE;
				bTransferError := TRUE;
				nTransferErrorID := 18;
				nTransferState := 255;
			(* When B enabled WB must be back *)
			ELSIF bSideBEnabled AND NOT( (fWAxisTransferPosition-0.2) <= stWBAxis.NcToPlc.ActPos ) THEN
				bAutoTransferPartsToDrill := FALSE;
				bTransferError := TRUE;
				nTransferErrorID := 19;
				nTransferState := 255;
			(* W Axis checked Ok *)
			ELSE
				nTransferAutoStep:=32;
			END_IF

		32: (* Initiate U Axis Move *)
			bUnloadPartsConfirmed:=FALSE;
			bTransferAxisMove := TRUE;
			fTransferMovePosition := fUAxisUnloadSidePosition;
			bAutoTransferWatchdog:=TRUE;
			tAutoTransferWatchdogTime := t#60s;
			nTransferAutoStep:=33;
			IF nCellRunoutCounter>=1 THEN
				nCellRunoutCounter:= nCellRunoutCounter-1;
			END_IF

		33: (* Wait for Move Done *)
			(* Move did not complete in time *)
			IF fbAutoTransferWatchdog.Q THEN
				bAutoTransferWatchdog:=FALSE;
				bTransferAxisMove := FALSE;
				bTransferError := TRUE;
				nTransferErrorID := 4;
				nTransferState := 254; (* Issue a stop *)
			(* Fault - Move Error *)
			ELSIF fbTransferAxisMove.Error THEN
				bAutoTransferWatchdog:=FALSE;
				bTransferAxisMove := FALSE;
				bTransferError := TRUE;
				nTransferErrorID := 5;
				nTransferState := 254; (* Issue a stop *)
			(* Move Done*)
			ELSIF bTransferAxisMove AND fbTransferAxisMove.Done THEN
				bAutoTransferPartsToDrill := FALSE;
				bAutoTransferWatchdog:=FALSE;
				bTransferAxisMove := FALSE;
				IF bCellRunoutRequest AND nCellRunoutCounter=1 THEN
					nTransferAutoStep:=40;
				ELSE
					nTransferAutoStep:=2;
				END_IF
			END_IF

		(* Lower Transfer *)
		40: (* Check Position of the Transfer *)
			IF bProx517 AND bProx516 THEN
				bTransferError := TRUE;
				nTransferErrorID := 3;
				nTransferState := 255;
			(* May want to check Transfer Position at Unload *)
			(* Checks OK *)
			ELSE
				bAutoRaise:= FALSE;
				nTransferAutoStep:=41;
			END_IF

		41: (* Lower Transfer *)
			bAutoLower:= TRUE;
			bAutoTransferWatchdog:=TRUE;
			tAutoTransferWatchdogTime := t#30s;
			(* Fault - Lower did not complete in time *)
			IF fbAutoTransferWatchdog.Q THEN
				bAutoTransferWatchdog:=FALSE;
				bTransferError := TRUE;
				nTransferErrorID := 6;
				nTransferState := 255;
			(* Down - Go to Move *)
			ELSIF fbProx517TON.Q  THEN
				bAutoTransferWatchdog:=FALSE;
				nTransferAutoStep:=nTransferAutoStep+1;
			END_IF

		42:(* Check that parts made it to Side A unload positions *)
			IF bSideADrilledParts THEN
				IF (sLoadSideSet = 'A') THEN
					(* Parts Missing on A side of Unload *)
					IF NOT(bProx510 AND bProx511 AND bProx512) THEN
						(* Fault - Parts missing on A side of Unload *)
						bTransferError := TRUE;
						nTransferErrorID := 10;
						nTransferState := 255;
						(* Clear both side tracking because we are asking for Operator Intervention *)
						bSideADrilledParts:=FALSE;
						bSideBDrilledParts:=FALSE;
					ELSE
						bSideADrilledParts:=FALSE;
						nTransferAutoStep:=nTransferAutoStep+1;
					END_IF
				ELSIF (sLoadSideSet = 'B') THEN
					(* Parts Missing on A side of Unload *)
					IF NOT(bProx410 AND bProx411 AND bProx412) THEN
						(* Fault - Parts missing on A side of Unload *)
						bTransferError := TRUE;
						nTransferErrorID := 10;
						nTransferState := 255;
						(* Clear both side tracking because we are asking for Operator Intervention *)
						bSideADrilledParts:=FALSE;
						bSideBDrilledParts:=FALSE;
					ELSE
						bSideADrilledParts:=FALSE;
						nTransferAutoStep:=nTransferAutoStep+1;
					END_IF
				END_IF
			(* Drilled Parts were not transfered for Side A, so check Side B *)
			ELSE
				nTransferAutoStep:=nTransferAutoStep+1;
			END_IF

		43:(* Check that parts made it to unload positions *)
			IF bSideBDrilledParts THEN
				IF (sLoadSideSet = 'A') THEN
					(* Parts Missing on B side of Unload *)
					IF NOT(bProx513 AND bProx514 AND bProx515) THEN
						(* Fault - Parts missing on B side of unload *)
						bTransferError := TRUE;
						nTransferErrorID := 15;
						nTransferState := 255;
						bSideBDrilledParts:=FALSE;
					ELSE
						bSideBDrilledParts:=FALSE;
						nTransferAutoStep:=50;
					END_IF
				ELSIF (sLoadSideSet = 'B') THEN
					(* Parts Missing on B side of Unload *)
					IF NOT(bProx413 AND bProx414 AND bProx415) THEN
						(* Fault - Parts missing on A side of Unload *)
						bTransferError := TRUE;
						nTransferErrorID := 15;
						nTransferState := 255;
						bSideBDrilledParts:=FALSE;
					ELSE
						bSideBDrilledParts:=FALSE;
						nTransferAutoStep:=50;
					END_IF
				END_IF
			(* Drilled Parts were not transfered for Side B, Move on *)
			ELSE
				nTransferAutoStep:=50;
			END_IF;

		(* Transfer to Load Position *)
		50: (* Trigger Move *)
			bTransferAxisMove := TRUE;
			fTransferMovePosition := fUAxisLoadSidePosition;
			bAutoTransferWatchdog:=TRUE;
			tAutoTransferWatchdogTime := t#60s;
			nTransferAutoStep:=51;

		51: (* Wait for Move Done *)
			(* Fault - Move did not complete in time *)
			IF fbAutoTransferWatchdog.Q THEN
				bAutoTransferWatchdog:=FALSE;
				bTransferAxisMove := FALSE;
				bTransferError := TRUE;
				nTransferErrorID := 4;
				nTransferState := 254; (* Issue a Stop *)
			(* Fault - Move Error *)
			ELSIF fbTransferAxisMove.Error THEN
				bAutoTransferWatchdog:=FALSE;
				bTransferAxisMove := FALSE;
				bTransferError := TRUE;
				nTransferErrorID := 5;
				nTransferState := 254; (* Issue a Stop *)
			(* Move Done*)
			ELSIF fbTransferAxisMove.Done THEN
				bAutoTransferWatchdog:=FALSE;
				bTransferAxisMove := FALSE;
				nTransferAutoStep:=2;
			END_IF

		END_CASE (* nTransferAutoStep *)


	254: (* Stop U Axis *)
		(* This step is necessary so we turn off the move command in a seperate scan of the program
		 than we turn on the stop command *)
		bUStop:=TRUE;
		bAutoTransferWatchdog:=TRUE;
		tAutoTransferWatchdogTime := t#1s;
		IF fbUAxisStop.Done OR fbAutoTransferWatchdog.Q THEN
			bUStop:=FALSE;
			bAutoTransferWatchdog:=FALSE;
			IF bTransferError THEN
				nTransferState:=255;
			ELSE
				nTransferState:=0;
			END_IF
		END_IF


	255: (* Fault State *)
		(* When in Auto Mode *)
		IF bMachineMode THEN
			(* Require that the fault be reset by the push button *)
			IF bFaultResetPB OR fbCommonFautlResetTON.Q THEN
				bTransferError := FALSE;
			END_IF
			(* When the error has been reset display "Press Cycle Start" *)
			IF  NOT bTransferError THEN
					bDispPressCycleStart:=TRUE;
				(* We want to wait for the Cycle Start to activate the transfer again. *)
				IF  MAIN.bCycleStartControlEnable THEN
					bDispPressCycleStart:=FALSE;
					(* When the transfer auto step is > 40 we want to go back to that step *)
					IF nTransferAutoStep < 40 THEN
						(* Otherwise we want to return step 2 to see what to do next *)
						nTransferAutoStep:=2;
					END_IF
					nTransferState := 2;
				END_IF
			END_IF
		(* In Manual we just jump back *)
		ELSE
			bTransferError := FALSE;
			nTransferState := 0;
			nTransferManualStep:=0;
		END_IF


	END_CASE	(* nTransferState *)

ELSE (* Reset all State Counters *)
	bAutoRaise := FALSE;
	bAutoLower := FALSE;
	nTransferState:=0;
	nTransferManualStep:=0;
	nTransferAutoStep:=0;
	bCellRunoutRequest:= FALSE;

END_IF

fbMoveToUnloadRTrig(CLK:=bAutoTransferPartsToDrill);
fbDownAndLoadRTrig(CLK:=bAutoTransferDownAndLoad AND NOT bFaultResetPB AND NOT fbCommonFautlResetTON.Q);
fbAutoTransferWatchdog(IN:=bAutoTransferWatchdog, PT:= tAutoTransferWatchdogTime);
fbUAxisStopTrig(CLK:= NOT(bMachineMode AND bInCycle) );
fbCellRunoutTrig(CLK:=bCellRunoutPB);

(* The bError bit will be on for one cycle when triggered and then will be reset the next scan in step 255 of the FB
So we want to translate into a text string from the error code *)
IF bTransferError THEN
	CASE nTransferErrorID OF
	01: sTransferErrorText := '01 - Load Side Must be Clear of Parts';
	02: sTransferErrorText := '02 - Transfer Did Not Raise In Time';
	03: sTransferErrorText := '03 - Transfer Raise-Lower Proxes All On';
	04: sTransferErrorText := '04 - Transfer Move Took To Long';
	05: sTransferErrorText := '05 - Transfer Move Command Failure';
	06: sTransferErrorText := '06 - Transfer Did Not Lower In Time';
	07: sTransferErrorText := '07 - W and X Axis Must be Homed';
	08: sTransferErrorText := '08 - Load Proxs Still Indicate Parts';
	09: sTransferErrorText := '09 - Transfer Must be Up to Move to Drill';
	10: sTransferErrorText := '10 - Parts Missing at Side A of Unload';
	11: sTransferErrorText := '11 - Side A Disabled, Remove Parts';
	12: sTransferErrorText := '12 - Side A Parts Missing on the Load Side';
	13: sTransferErrorText := '13 - Side B Disabled, Remove Parts';
	14: sTransferErrorText := '14 - Side B Parts Missing on the Load Side';
	15: sTransferErrorText := '15 - Parts Missing at Side B of Unload';
	16: sTransferErrorText := '16 - Transfer Must be at Load Position';
	17: sTransferErrorText := '17 - Unload Side Must be Clear of Parts';
	18: sTransferErrorText := '18 - WA Axis to far Forward to Transfer';
	19: sTransferErrorText := '19 - WB Axis to far Forward to Transfer';

	(* Errors > 50 are handled as Faults by the Program and Kick out of Auto *)
	50: sTransferErrorText := '00 - Transfer Must be at Load Position to go into Auto';
	51: sTransferErrorText := '01 -  X Axis Must be Homed to go into Auto';
	52: sTransferErrorText := '02 - Transfer Must be Down to go into Auto';
	53: sTransferErrorText := '03 - W and X Axis Must be Homed to go into Auto';
	54: sTransferErrorText := '04 - Transfer Raise and Lower Proxes On At Same Time';
	END_CASE
END_IF
END_ACTION

(* POU Programs/P_TailstockControl, ST *)
PROGRAM P_TailstockControl
VAR
(* WA Axis MC Functions *)
	fbWAAxisPower: MC_Power;
	fbWAAxisMove: MC_MoveAbsolute;
	fbWAAxisSetZero: MC_SetPosition;
	bWAAxisPower: BOOL := FALSE;
	bWAAxisMove: BOOL := FALSE;
	bWAAxisSetZero: BOOL := FALSE;
	fWAAxisSetZeroPosition: LREAL := 0.0;
	bWADeCtrlEnable : BOOL := FALSE;		(* Enable bit for FB to move off overtravel *)
	fbHomeWAPBRTrig : R_TRIG;			(* Capture the Rising Edge of the PB *)

(* WB Axis MC Functions *)
	fbWBAxisPower: MC_Power;
	fbWBAxisMove: MC_MoveAbsolute;
	fbWBAxisSetZero: MC_SetPosition;
	bWBAxisPower: BOOL := FALSE;
	bWBAxisMove: BOOL := FALSE;
	bWBAxisSetZero: BOOL := FALSE;
	fWBAxisSetZeroPosition: LREAL := 0.0;
	bWBDeCtrlEnable : BOOL := FALSE;		(* Enable bit for FB to move off overtravel *)
	fbHomeWBPBRTrig : R_TRIG;			(* Capture the Rising Edge of the PB *)

	bTransferAtPosition: BOOL := FALSE;			(* Transfer is at Load or unload position *)

	bAManualOpenCollet: BOOL := FALSE;		(*Manual Control to Open the Collets on Side A*)
	bAManualCloseCollet: BOOL := FALSE;		(*Manual Control to Close the Collets on Side A*)
	bBManualOpenCollet: BOOL := FALSE;		(*Manual Control to Open the Collets on Side B*)
	bBManualCloseCollet: BOOL := FALSE;		(*Manual Control to Close the Collets on Side B*)

(* Recording Variables *)
	nWAThrustMaxRecorded: DINT := 0;						(* Recorded Max thrust value seen on WA Axis*)
	arraynWAThrustMaxRec: ARRAY [1..20] OF DINT :=20(0);	(* Store the Values of the last 10 runs for WA *)
	nWBThrustMaxRecorded: DINT := 0;						(* Recorded Max thrust value seen on WB Axis *)
	arraynWBThrustMaxRec: ARRAY [1..20] OF DINT :=20(0);	(* Store the Values of the last 10 runs for WB *)
	fbStoreWMaxThrust: R_TRIG;							(* Trigger to stroe the values *)
	nUThrustMaxRecorded: DINT := 0;						(* Recorded Max thrust value seen on U Axis *)


END_VAR
(* Call Actions *)
Tailstock_Function;
(* Check Transfer at Load or Unload Positions *)
bTransferAtPosition:=
	(* Within +/- 0.1mm of Unload position *)
	( (fUAxisUnloadSidePosition+0.1)>=stUAxis.NcToPlc.ActPos AND
	stUAxis.NcToPlc.ActPos>=(fUAxisUnloadSidePosition-0.1) ) OR
	(* Within +/- 0.1mm of Load position *)
	( (fUAxisLoadSidePosition+0.1)>=stUAxis.NcToPlc.ActPos AND
	stUAxis.NcToPlc.ActPos>=(fUAxisLoadSidePosition-0.1) );

(* Turn on MC_Power when Hard Enable is ON *)
bWAAxisPower := bAServoEnable;
bWBAxisPower := bBServoEnable;

fbWAAxisPower(
	Enable:=bWAAxisPower ,
	Enable_Positive:= bWAAxisPower ,
	Enable_Negative:= bWAAxisPower ,
	Override:=100 ,
	BufferMode:=MC_Aborting ,
	Axis:=stWAAxis );

(* When the Stop is Done or has an error then we turn off the trigger *)
IF fbWAAxisStop.Done OR fbWAAxisStop.Error THEN
	bWAStop:=FALSE;
END_IF
fbWAAxisStop(
	Execute := bWAStop,
	Deceleration := 0,
	Jerk := 0,
	Axis := stWAAxis );

fbWAAxisMCReset(
	Execute:=bWAMCResetRequest ,
	Axis:=stWAAxis );

fbWAAxisDriveReset(
	NetId:='' ,
	Execute:=bZWADriveResetRequest ,
	Timeout:=t#10s ,
	Axis:= stWAAxis, );

stWAAxis.ReadStatus();

(* If a Drive reset was requested then when the Drive Reset is done we want to do a MC Reset of the NC Axis *)
IF bZWADriveResetRequest AND (NOT (fbWAAxisDriveReset.Busy) OR  fbWAAxisDriveReset.Error) THEN
	bWAMCResetRequest:=TRUE;
END_IF
IF fbWAAxisMCReset.Done OR fbWAAxisMCReset.Error THEN
	bWAMCResetRequest:=FALSE;
	bZWADriveResetRequest:=FALSE;
END_IF

(* When the Home PB pressed trigger a home *)
fbHomeWAPBRTrig(CLK:=bWAAxisHomePB);
IF fbHomeWAPBRTrig.Q  AND NOT bMachineFault THEN
	bWAAxisHome:=TRUE;
(* When Home is done turn off trigger *)
ELSIF fbWAAxisHome.Done THEN
	bWAAxisHome:=FALSE;
(* if an Error then issue a stop *)
ELSIF  fbWAAxisHome.Error THEN
	bWAAxisHome:=FALSE;
	bWAStop:=TRUE;
END_IF

(* Home WA Axis *)
fbWAAxisHome(
	Execute:= bWAAxisHome,
	Position:= fWAAxisHomeOffset ,
	HomingMode:= ,
	BufferMode:= ,
	Options:= ,
	bCalibrationCam:= DriveZAWAdinputs.6 ,
	Axis:= stWAAxis ,
	Done=> ,
	Busy=> ,
	Active=> ,
	CommandAborted=> ,
	Error=> ,
	ErrorID=>  );

(* If one of the WA Axis overtravel limit switches is made, then turn on the bit that allows
Movement off of the limit switchs *)
IF NOT(DriveZAWAdinputs.3) OR NOT(DriveZAWAdinputs.4) THEN
	bWADeCtrlEnable:=TRUE;
ELSE
	bWADeCtrlEnable:=FALSE;
END_IF
stWAAxis.PlcToNc.ControlDWord :=
AxisSetAcceptBlockedDriveSignal(stWAAxis.PlcToNc.ControlDWord,
	bEnable:= bWADeCtrlEnable );


(*	SIDE B 	*)
bBServoEnable;		(* Display the B Sode Enable Relay for Convenience *)

fbWBAxisPower(
	Enable:= bWBAxisPower ,
	Enable_Positive:= bWBAxisPower ,
	Enable_Negative:= bWBAxisPower ,
	Override:=100 ,
	BufferMode:=MC_Aborting ,
	Axis:=stWBAxis );

(* When the Stop is Done or has an error then we turn off the trigger *)
IF fbWBAxisStop.Done OR fbWBAxisStop.Error THEN
	bWBStop:=FALSE;
END_IF
fbWBAxisStop(
	Execute := bWBStop,
	Deceleration := 0,
	Jerk := 0,
	Axis := stWBAxis );

fbWBAxisMCReset(
	Execute:=bWBMCResetRequest ,
	Axis:=stWBAxis );

fbWBAxisDriveReset(
	NetId:='' ,
	Execute:=bZWBDriveResetRequest ,
	Timeout:=t#10s ,
	Axis:= stWBAxis, );

stWBAxis.ReadStatus();

(* If a Drive reset was requested then when the Drive Reset is done we want to do a MC Reset of the NC Axis *)
IF bZWBDriveResetRequest AND (NOT (fbWBAxisDriveReset.Busy) OR  fbWBAxisDriveReset.Error) THEN
	bWBMCResetRequest:=TRUE;
END_IF
IF fbWBAxisMCReset.Done OR fbWBAxisMCReset.Error THEN
	bWBMCResetRequest:=FALSE;
	bZWBDriveResetRequest:=FALSE;
END_IF

(* When the Home PB pressed trigger a home *)
fbHomeWBPBRTrig(CLK:=bWBAxisHomePB);
IF fbHomeWBPBRTrig.Q AND NOT bMachineFault THEN
	bWBAxisHome:=TRUE;
(* When Home is done turn off trigger *)
ELSIF fbHomeWB.Done THEN
	bWBAxisHome:=FALSE;	(* Also set True from MM_HomeAutomation *)
(* If an error occurs issue a stop *)
ELSIF fbHomeWB.Error THEN
	bWBAxisHome:=FALSE;
	bWBStop:=TRUE;
END_IF

(* Home WB Axis *)
fbHomeWB(
	Execute:= bWBAxisHome,
	Position:= fWBAxisHomeOffset ,
	HomingMode:= ,
	BufferMode:= ,
	Options:= ,
	bCalibrationCam:= DriveZBWBdinputs.6 ,
	Axis:= stWBAxis ,
	Done=> ,
	Busy=> ,
	Active=> ,
	CommandAborted=> ,
	Error=> ,
	ErrorID=> );

(* If one of the WB Axis overtravel limit switches is made, then turn on the bit that allows
Movement off of the limit switchs *)
IF NOT(DriveZBWBdinputs.3) OR NOT(DriveZBWBdinputs.4) THEN
	bWBDeCtrlEnable:=TRUE;
ELSE
	bWBDeCtrlEnable:=FALSE;
END_IF
stWBAxis.PlcToNc.ControlDWord :=
AxisSetAcceptBlockedDriveSignal(stWBAxis.PlcToNc.ControlDWord,
	bEnable:= bWBDeCtrlEnable );

(* Assign the Ejectors State *)
nAEjectorAdvancedState.0:=bProx613;
nAEjectorAdvancedState.1:=bProx614;
nAEjectorAdvancedState.2:=bProx615;
nAEjectorRetractedState.0:=bProx610;
nAEjectorRetractedState.1:=bProx611;
nAEjectorRetractedState.2:=bProx612;

nBEjectorAdvancedState.0:=bProx723;
nBEjectorAdvancedState.1:=bProx724;
nBEjectorAdvancedState.2:=bProx725;
nBEjectorRetractedState.0:=bProx720;
nBEjectorRetractedState.1:=bProx721;
nBEjectorRetractedState.2:=bProx722;



(*	******* COLLET CLAMP ******	*)
(* Side A *)
(* Fire Solenoid Valves *)
(* Normal Control is handled in the FB_Fixture Control *)
(* When the MCR is off we turn off the solenoids *)
IF NOT (bMCR AND bHydraulicPowerUnitRunning) THEN
	bATailstockColletUnclamp := FALSE;
	bATailstockColletClamp:=FALSE;
END_IF
(*FAIL-SAFE CONTROL
If Both Outputs are on at the same time then turn them Off and Fault *)
IF bATailstockColletUnclamp AND bATailstockColletClamp THEN
	nModeError:=Er_SideAColletSolError;
	bATailstockColletUnclamp := FALSE;
	bATailstockColletClamp:=FALSE;
END_IF

(* Side B *)
(* Fire Solenoid Valves *)
(* Normal Control is handled in the FB_Fixture Control *)
(* When the MCR is off we turn off the solenoids *)
IF NOT (bMCR AND bHydraulicPowerUnitRunning) THEN
	bBTailstockColletUnclamp := FALSE;
	bBTailstockColletClamp:=FALSE;
END_IF
(*FAIL-SAFE CONTROL
If Both Outputs are on at the same time then turn them Off and Fault *)
IF bBTailstockColletUnclamp AND bBTailstockColletClamp THEN
	nModeError:=Er_SideBColletSolError;
	bBTailstockColletUnclamp := FALSE;
	bBTailstockColletClamp:=FALSE;
END_IF

(*	******* EJECTORS  ******	*)
(* Side A *)
(* Fire Solenoid Valves *)
(* Normal Control is handled in the FB_Fixture Control *)
(* If MCR off or Air Pressure Lost *)
IF NOT (bMCR AND bPneumaticSystemPressure) THEN
	bAEjectorsAdvance := FALSE;
	bAEjectorsRetract := FALSE;
END_IF
(*FAIL-SAFE CONTROL
If Both Outputs are on at the same time then turn them Off and Fault *)
IF bAEjectorsAdvance AND bAEjectorsRetract THEN
	nModeError:=Er_SideAEjectorsSolError;
	bAEjectorsAdvance := FALSE;
	bAEjectorsRetract := FALSE;
END_IF

(* Side B *)
(* Fire Solenoid Valves *)
(* Normal Control is handled in the FB_Fixture Control *)
(* If MCR off or Air Pressure Lost *)
IF NOT (bMCR AND bPneumaticSystemPressure) THEN
	bBEjectorsAdvance := FALSE;
	bBEjectorsRetract := FALSE;
END_IF
(*FAIL-SAFE CONTROL
If Both Outputs are on at the same time then turn them Off and Fault *)
IF bBEjectorsAdvance AND bBEjectorsRetract THEN
	nModeError:=Er_SideBEjectorsSolError;
	bBEjectorsAdvance := FALSE;
	bBEjectorsRetract := FALSE;
END_IF

(* Fault if Manual Move Pressed *)
IF (bWAAxisAdvancePB OR bWAAxisRetractPB) AND
	bMPGAOn
THEN
	nModeError:=Er_MPG_A_Active;
END_IF
IF (bWBAxisAdvancePB OR bWBAxisRetractPB) AND
	bMPGBOn
THEN
	nModeError:=Er_MPG_B_Active;
END_IF


(* Record W Axis Thrust *)
	(* Reset the W Thrust before Drilling *)
(*	IF nAutoCycleStep = AC_SpindleOn THEN
		nWAThrustMaxRecorded:=0;
		nWBThrustMaxRecorded:=0;
	END_IF
*)
	(* Record Max WA Thrust  while in the Clamp State*)
	IF nWAAxisThrust > nWAThrustMaxRecorded AND nAutoCycleStep=AC_Clamp THEN
		nWAThrustMaxRecorded:=nWAAxisThrust;
	END_IF
	(* Record Max WB Thrust *)
	IF nWBAxisThrust > nWBThrustMaxRecorded AND nAutoCycleStep=AC_Clamp THEN
		nWBThrustMaxRecorded:=nWBAxisThrust;
	END_IF
	(* Record Max U Axis Thrust *)
	IF nUAxisThrust > nUThrustMaxRecorded THEN
		nUThrustMaxRecorded:=nUAxisThrust;
	END_IF

(* Store the value in the array when we are done drilling *)
fbStoreWMaxThrust(CLK:=nAutoCycleStep=AC_SpindleOff);
IF fbStoreWMaxThrust.Q THEN
	arraynWAThrustMaxRec[20]	:=arraynWAThrustMaxRec[19];
	arraynWAThrustMaxRec[19]	:=arraynWAThrustMaxRec[18];
	arraynWAThrustMaxRec[18]	:=arraynWAThrustMaxRec[17];
	arraynWAThrustMaxRec[17]	:=arraynWAThrustMaxRec[16];
	arraynWAThrustMaxRec[16]	:=arraynWAThrustMaxRec[15];
	arraynWAThrustMaxRec[15]	:=arraynWAThrustMaxRec[14];
	arraynWAThrustMaxRec[14]	:=arraynWAThrustMaxRec[13];
	arraynWAThrustMaxRec[13]	:=arraynWAThrustMaxRec[12];
	arraynWAThrustMaxRec[12]	:=arraynWAThrustMaxRec[11];
	arraynWAThrustMaxRec[11]	:=arraynWAThrustMaxRec[10];
	arraynWAThrustMaxRec[10]	:=arraynWAThrustMaxRec[9];
	arraynWAThrustMaxRec[9]		:=arraynWAThrustMaxRec[8];
	arraynWAThrustMaxRec[8]		:=arraynWAThrustMaxRec[7];
	arraynWAThrustMaxRec[7]		:=arraynWAThrustMaxRec[6];
	arraynWAThrustMaxRec[6]		:=arraynWAThrustMaxRec[5];
	arraynWAThrustMaxRec[5]		:=arraynWAThrustMaxRec[4];
	arraynWAThrustMaxRec[4]		:=arraynWAThrustMaxRec[3];
	arraynWAThrustMaxRec[3]		:=arraynWAThrustMaxRec[2];
	arraynWAThrustMaxRec[2]		:=arraynWAThrustMaxRec[1];
	arraynWAThrustMaxRec[1]		:=nWAThrustMaxRecorded;
	nWAThrustMaxRecorded		:=0;	(* Reset Variable *)

	arraynWBThrustMaxRec[20]	:=arraynWBThrustMaxRec[19];
	arraynWBThrustMaxRec[19]	:=arraynWBThrustMaxRec[18];
	arraynWBThrustMaxRec[18]	:=arraynWBThrustMaxRec[17];
	arraynWBThrustMaxRec[17]	:=arraynWBThrustMaxRec[16];
	arraynWBThrustMaxRec[16]	:=arraynWBThrustMaxRec[15];
	arraynWBThrustMaxRec[15]	:=arraynWBThrustMaxRec[14];
	arraynWBThrustMaxRec[14]	:=arraynWBThrustMaxRec[13];
	arraynWBThrustMaxRec[13]	:=arraynWBThrustMaxRec[12];
	arraynWBThrustMaxRec[12]	:=arraynWBThrustMaxRec[11];
	arraynWBThrustMaxRec[11]	:=arraynWBThrustMaxRec[10];
	arraynWBThrustMaxRec[10]	:=arraynWBThrustMaxRec[9];
	arraynWBThrustMaxRec[9]		:=arraynWBThrustMaxRec[8];
	arraynWBThrustMaxRec[8]		:=arraynWBThrustMaxRec[7];
	arraynWBThrustMaxRec[7]		:=arraynWBThrustMaxRec[6];
	arraynWBThrustMaxRec[6]		:=arraynWBThrustMaxRec[5];
	arraynWBThrustMaxRec[5]		:=arraynWBThrustMaxRec[4];
	arraynWBThrustMaxRec[4]		:=arraynWBThrustMaxRec[3];
	arraynWBThrustMaxRec[3]		:=arraynWBThrustMaxRec[2];
	arraynWBThrustMaxRec[2]		:=arraynWBThrustMaxRec[1];
	arraynWBThrustMaxRec[1]		:=nWBThrustMaxRecorded;
	nWBThrustMaxRecorded		:=0;	(* Reset Variable *)
END_IF
END_PROGRAM
ACTION Tailstock_Function:
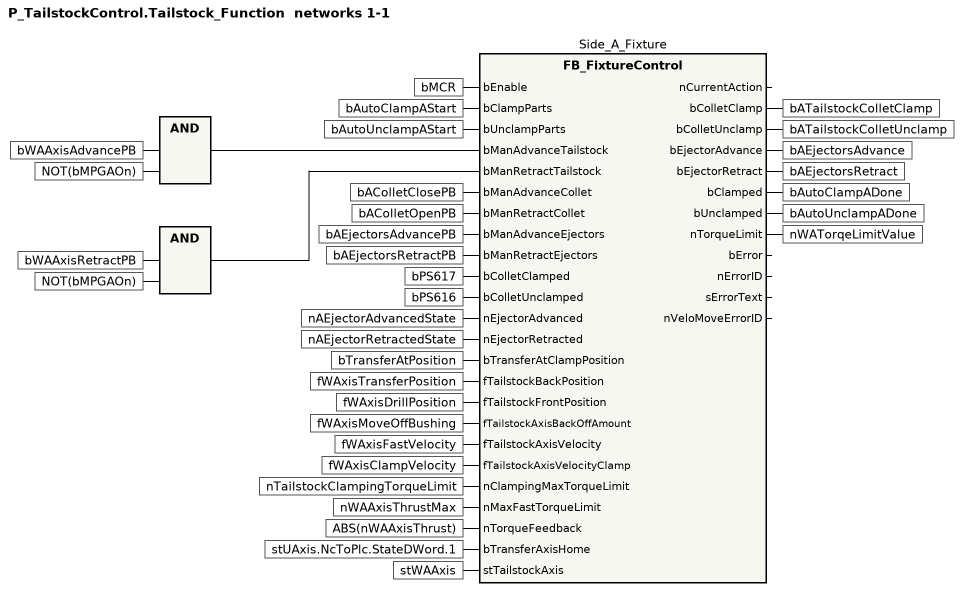
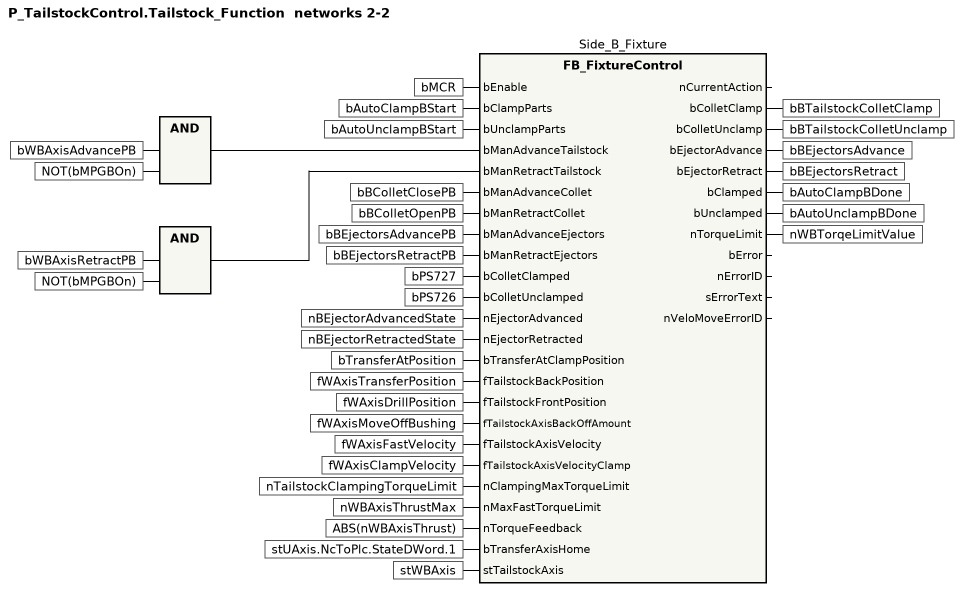
_FBD_ (* Function Block Diagram *)
NETWORK 1
	Side_A_Fixture:FB_FixtureControl(bEnable: bMCR, bClampParts: bAutoClampAStart, bUnclampParts: bAutoUnclampAStart, bManAdvanceTailstock: AND(bWAAxisAdvancePB, NOT(bMPGAOn)), bManRetractTailstock: AND(bWAAxisRetractPB, NOT(bMPGAOn)), bManAdvanceCollet: bAColletClosePB, bManRetractCollet: bAColletOpenPB, bManAdvanceEjectors: bAEjectorsAdvancePB, bManRetractEjectors: bAEjectorsRetractPB, bColletClamped: bPS617, bColletUnclamped: bPS616, nEjectorAdvanced: nAEjectorAdvancedState, nEjectorRetracted: nAEjectorRetractedState, bTransferAtClampPosition: bTransferAtPosition, fTailstockBackPosition: fWAxisTransferPosition, fTailstockFrontPosition: fWAxisDrillPosition, fTailstockAxisBackOffAmount: fWAxisMoveOffBushing, fTailstockAxisVelocity: fWAxisFastVelocity, fTailstockAxisVelocityClamp: fWAxisClampVelocity, nClampingMaxTorqueLimit: nTailstockClampingTorqueLimit, nMaxFastTorqueLimit: nWAAxisThrustMax, nTorqueFeedback: ABS(nWAAxisThrust), bTransferAxisHome: stUAxis.NcToPlc.StateDWord.1, stTailstockAxis: stWAAxis, bColletClamp => bATailstockColletClamp, bColletUnclamp => bATailstockColletUnclamp, bEjectorAdvance => bAEjectorsAdvance, bEjectorRetract => bAEjectorsRetract, bClamped => bAutoClampADone, bUnclamped => bAutoUnclampADone, nTorqueLimit => nWATorqeLimitValue)
NETWORK 2
	Side_B_Fixture:FB_FixtureControl(bEnable: bMCR, bClampParts: bAutoClampBStart, bUnclampParts: bAutoUnclampBStart, bManAdvanceTailstock: AND(bWBAxisAdvancePB, NOT(bMPGBOn)), bManRetractTailstock: AND(bWBAxisRetractPB, NOT(bMPGBOn)), bManAdvanceCollet: bBColletClosePB, bManRetractCollet: bBColletOpenPB, bManAdvanceEjectors: bBEjectorsAdvancePB, bManRetractEjectors: bBEjectorsRetractPB, bColletClamped: bPS727, bColletUnclamped: bPS726, nEjectorAdvanced: nBEjectorAdvancedState, nEjectorRetracted: nBEjectorRetractedState, bTransferAtClampPosition: bTransferAtPosition, fTailstockBackPosition: fWAxisTransferPosition, fTailstockFrontPosition: fWAxisDrillPosition, fTailstockAxisBackOffAmount: fWAxisMoveOffBushing, fTailstockAxisVelocity: fWAxisFastVelocity, fTailstockAxisVelocityClamp: fWAxisClampVelocity, nClampingMaxTorqueLimit: nTailstockClampingTorqueLimit, nMaxFastTorqueLimit: nWBAxisThrustMax, nTorqueFeedback: ABS(nWBAxisThrust), bTransferAxisHome: stUAxis.NcToPlc.StateDWord.1, stTailstockAxis: stWBAxis, bColletClamp => bBTailstockColletClamp, bColletUnclamp => bBTailstockColletUnclamp, bEjectorAdvance => bBEjectorsAdvance, bEjectorRetract => bBEjectorsRetract, bClamped => bAutoClampBDone, bUnclamped => bAutoUnclampBDone, nTorqueLimit => nWBTorqeLimitValue)
_END_FBD_
(* the same logic as Structured Text *)
(* Network 1 *)
Side_A_Fixture(bEnable := bMCR, bClampParts := bAutoClampAStart, bUnclampParts := bAutoUnclampAStart, bManAdvanceTailstock := bWAAxisAdvancePB AND NOT(bMPGAOn), bManRetractTailstock := bWAAxisRetractPB AND NOT(bMPGAOn), bManAdvanceCollet := bAColletClosePB, bManRetractCollet := bAColletOpenPB, bManAdvanceEjectors := bAEjectorsAdvancePB, bManRetractEjectors := bAEjectorsRetractPB, bColletClamped := bPS617, bColletUnclamped := bPS616, nEjectorAdvanced := nAEjectorAdvancedState, nEjectorRetracted := nAEjectorRetractedState, bTransferAtClampPosition := bTransferAtPosition, fTailstockBackPosition := fWAxisTransferPosition, fTailstockFrontPosition := fWAxisDrillPosition, fTailstockAxisBackOffAmount := fWAxisMoveOffBushing, fTailstockAxisVelocity := fWAxisFastVelocity, fTailstockAxisVelocityClamp := fWAxisClampVelocity, nClampingMaxTorqueLimit := nTailstockClampingTorqueLimit, nMaxFastTorqueLimit := nWAAxisThrustMax, nTorqueFeedback := ABS(nWAAxisThrust), bTransferAxisHome := stUAxis.NcToPlc.StateDWord.1, stTailstockAxis := stWAAxis);
bATailstockColletClamp := Side_A_Fixture.bColletClamp;
bATailstockColletUnclamp := Side_A_Fixture.bColletUnclamp;
bAEjectorsAdvance := Side_A_Fixture.bEjectorAdvance;
bAEjectorsRetract := Side_A_Fixture.bEjectorRetract;
bAutoClampADone := Side_A_Fixture.bClamped;
bAutoUnclampADone := Side_A_Fixture.bUnclamped;
nWATorqeLimitValue := Side_A_Fixture.nTorqueLimit;
(* Network 2 *)
Side_B_Fixture(bEnable := bMCR, bClampParts := bAutoClampBStart, bUnclampParts := bAutoUnclampBStart, bManAdvanceTailstock := bWBAxisAdvancePB AND NOT(bMPGBOn), bManRetractTailstock := bWBAxisRetractPB AND NOT(bMPGBOn), bManAdvanceCollet := bBColletClosePB, bManRetractCollet := bBColletOpenPB, bManAdvanceEjectors := bBEjectorsAdvancePB, bManRetractEjectors := bBEjectorsRetractPB, bColletClamped := bPS727, bColletUnclamped := bPS726, nEjectorAdvanced := nBEjectorAdvancedState, nEjectorRetracted := nBEjectorRetractedState, bTransferAtClampPosition := bTransferAtPosition, fTailstockBackPosition := fWAxisTransferPosition, fTailstockFrontPosition := fWAxisDrillPosition, fTailstockAxisBackOffAmount := fWAxisMoveOffBushing, fTailstockAxisVelocity := fWAxisFastVelocity, fTailstockAxisVelocityClamp := fWAxisClampVelocity, nClampingMaxTorqueLimit := nTailstockClampingTorqueLimit, nMaxFastTorqueLimit := nWBAxisThrustMax, nTorqueFeedback := ABS(nWBAxisThrust), bTransferAxisHome := stUAxis.NcToPlc.StateDWord.1, stTailstockAxis := stWBAxis);
bBTailstockColletClamp := Side_B_Fixture.bColletClamp;
bBTailstockColletUnclamp := Side_B_Fixture.bColletUnclamp;
bBEjectorsAdvance := Side_B_Fixture.bEjectorAdvance;
bBEjectorsRetract := Side_B_Fixture.bEjectorRetract;
bAutoClampBDone := Side_B_Fixture.bClamped;
bAutoUnclampBDone := Side_B_Fixture.bUnclamped;
nWBTorqeLimitValue := Side_B_Fixture.nTorqueLimit;
END_ACTION

(* POU Function Blocks/FB_FixtureControl, ST *)
FUNCTION_BLOCK FB_FixtureControl
VAR_INPUT
	bEnable: BOOL;
	(* Command Inputs *)
	(***AUTOMATIC***)
	bClampParts: BOOL;			(* PRIORITY 1 *)
	bUnclampParts: BOOL;			(* PRIORITY 2 *)
	(***MANUAL***)
	bManAdvanceTailstock: BOOL;		(* PRIORITY 4 *)
	bManRetractTailstock: BOOL;		(* PRIORITY 5 *)
	bManAdvanceCollet: BOOL;		(* PRIORITY 6 *)
	bManRetractCollet: BOOL;			(* PRIORITY 7 *)
	bManAdvanceEjectors: BOOL;		(* PRIORITY 8 *)
	bManRetractEjectors: BOOL;		(* PRIORITY 9 *)

	(* Feedback Inputs *)
	bColletClamped: BOOL;		(* PS *)
	bColletUnclamped: BOOL;		(* PS *)
	nEjectorAdvanced: USINT;
	nEjectorRetracted: USINT;
	(* COMM Inputs *)
	bTransferAtClampPosition : BOOL;
	(* OTHER INPUTS *)
	fTailstockBackPosition: LREAL;
	fTailstockFrontPosition: LREAL;
	fTailstockAxisBackOffAmount: LREAL;
	fTailstockAxisVelocity: LREAL;			(* Speed for all moves but swallowing part *)
	fTailstockAxisVelocityClamp: LREAL;		(* Speed for move to swallow part *)
	nClampingMaxTorqueLimit: UDINT;		(* Max set value for the torque limit while moving to
 Position - Swallowing Part *)
	nMaxFastTorqueLimit: UDINT;			(* Max set value for the torque limit while moving all other moves *)
	nTorqueFeedback : INT ;
	bTransferAxisHome : BOOL;			(* Transfer Axis is homed *)
END_VAR
VAR_OUTPUT
	nCurrentAction: USINT := 0;
	(* Command Outputs *)
	bColletClamp: BOOL;
	bColletUnclamp: BOOL;
	bEjectorAdvance: BOOL;
	bEjectorRetract: BOOL;
	(* COMM Outputs *)
	bClamped: BOOL;
	bUnclamped: BOOL;
	nTorqueLimit: INT := 1000;			(* %, 0 - 1000 *)
	bError: BOOL;
	nErrorID: UDINT;
	(* We do not clear this string so we can see what the last error was through TwinCAT *)
	sErrorText: STRING := '';			(* Text string to be displayed for current error - Fault # Put in by program *)
	nVeloMoveErrorID: UDINT := 0;
END_VAR
VAR_IN_OUT
	stTailstockAxis: AXIS_REF;
END_VAR
VAR
	fTailstockLoadPositionOne: LREAL;		(* Delete This Position *)
	fbTailstockAxisPower: MC_Power;
	fbTailstockAxisHome: MC_Home;
	fbTailstockAxisMoveTo: MC_MoveAbsolute;
	fbTailstockAxisMoveVelo: MC_MoveVelocity;
	fbTailstockAxisStop: MC_Stop;
	bTailstockAxisPower: BOOL := FALSE;
	bTailstockAxisHome: BOOL := FALSE;
	bTailstockAxisMove: BOOL := FALSE;
	bTailstockAxisMoveVelo: BOOL := FALSE;
	fTailstockMoveVelo: LREAL := 10.0;
	fTailstockAxisPosition: LREAL := 0.0;
	bTailstockAxisSetZero: BOOL := FALSE;
	bTailstockAxisStop: BOOL := FALSE;

	nTorqueLimitRequest: INT;				(* % , 0 - 1000 *)(* Will need to be an input if start using *)

	nClampingState: USINT := 0;
	nUnclampingState: USINT := 0;

	fbColletClampTimeout: TON;
	fbClampOffTON: TON;						(* Timer to make sure the solenoid is de-energized *)
	fbColletUnclampTimeout: TON;
	fbUnclampOffTON: TON;					(* Timer to make sure the solenoid is de-energized *)
	fbEjectorAdvanceTimeout: TON;
	fbEjectAdvOffTON: TON;					(* Timer to make sure the solenoid is de-energized *)
	fbEjectorRetractTimeout: TON;
	fbEjectRetOffTON: TON;					(* Timer to make sure the solenoid is de-energized *)

	fbClampPartsRTRIG: R_TRIG;
	fbUnclampPartsRTRIG: R_TRIG;
	fbHomeTailstockAxisRTRIG: R_TRIG;
	fbAdvanceTailstockRTRIG: R_TRIG;
	fbRetractTailstockRTRIG: R_TRIG;
	fbAdvanceColletRTRIG: R_TRIG;
	fbRetractColletRTRIG: R_TRIG;
	fbAdvanceEjectorsRTRIG: R_TRIG;
	fbRetractEjectorsRTRIG: R_TRIG;
	fbColletClampTON: TON;
	fbEjectorAdvanceTON: TON;
	fbEjectorAdvanceT5TON: TON; (*Gives a Delay after last ejector comes off retracted prox., No hard sensor for this*)
	fbEjectorRetractTON: TON;
	fbColletUnclampTON: TON;
	bEjectorAdvanceTON: BOOL := FALSE;
	fbTorqueLimitTON: TON;
	bTorqueLimitTimeout: BOOL := FALSE;
	bColletClampTON: BOOL := FALSE;
	bEjectorRetractTON: BOOL := FALSE;
	bColletUnclampTON: BOOL := FALSE;
	fTailstockAxisVelocityLocal: LREAL;

	fbTogglePositionLagMonitoring: MC_WriteBoolParameter;
	fbPositionLagMonitingStatus : MC_ReadBoolParameter;
	bTogglePositionLagMonitoring: BOOL := FALSE;
	bPositionLagMonitoiring : BOOL;
	nTestCount: INT := 0;		(*Test Counter*)
END_VAR
CASE nCurrentAction OF
0:	(* Initial State *)
		bTailstockAxisStop:=FALSE;
		(* We need to reset the Torque Limit to 100% if we E-Stop or Fault to be ready for the next move *)
		nTorqueLimit := 1000;
	IF bEnable THEN
		nCurrentAction:=nCurrentAction+1;
	END_IF

1:(* A STEP TO CHECK FEED BACK DEVICES TO FIRE SOLENOIDS *)
	IF bColletClamped AND NOT(bColletUnclamped) THEN
		bColletUnclamp:=FALSE;
		bColletClamp:=TRUE;
	END_IF
	IF bColletUnclamped AND NOT(bColletClamped) THEN
		bColletUnclamp:=TRUE;
		bColletClamp:=FALSE;
	END_IF
	IF nEjectorAdvanced=7 AND NOT(nEjectorRetracted>0) THEN
		bEjectorAdvance:=TRUE;
		bEjectorRetract:=FALSE;
	END_IF
	IF nEjectorRetracted=7 AND nEjectorAdvanced=7 THEN
		bEjectorRetract:=TRUE;
		bEjectorAdvance:=FALSE;
	END_IF
	nCurrentAction:=nCurrentAction+1;

2: (* Alwasys return to this step to Wait for the next command *)
	IF NOT(bEnable) THEN
		bColletClamp:=FALSE;
		bColletUnclamp:=FALSE;
		bEjectorAdvance:=FALSE;
		bEjectorRetract:=FALSE;
		bTailstockAxisMove:=FALSE;
		bTailstockAxisMoveVelo:=FALSE;
		bTailstockAxisStop:=TRUE;
		nCurrentAction:=0;
	ELSIF fbClampPartsRTRIG.Q THEN
		nCurrentAction:=3;
	ELSIF fbUnclampPartsRTRIG.Q THEN
		nCurrentAction:=4;
	ELSIF fbAdvanceTailstockRTRIG.Q THEN
		nCurrentAction:=6;
	ELSIF fbRetractTailstockRTRIG.Q THEN
		nCurrentAction:=7;
	ELSIF fbAdvanceColletRTRIG.Q THEN
		nCurrentAction:=8;
	ELSIF fbRetractColletRTRIG.Q THEN
		nCurrentAction:=9;
	ELSIF fbAdvanceEjectorsRTRIG.Q THEN
		nCurrentAction:=10;
	ELSIF fbRetractEjectorsRTRIG.Q THEN
		nCurrentAction:=11;
	END_IF

